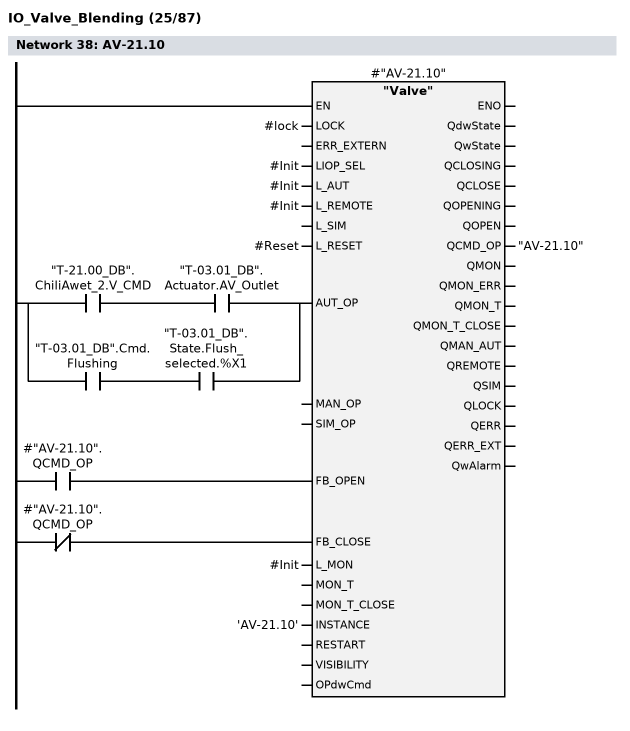
   RUNG wire#powerrail
      #"AV-21.10"(AUT_OP := wire#w1, FB_OPEN := wire#w2, FB_CLOSE := wire#w3, LOCK := #lock, ERR_EXTERN :=, LIOP_SEL := #Init, L_AUT := #Init, L_REMOTE := #Init, L_SIM :=, L_RESET := #Reset, MAN_OP :=, SIM_OP :=, L_MON := #Init, MON_T :=, MON_T_CLOSE :=, INSTANCE := 'AV-21.10', RESTART :=, VISIBILITY :=, OPdwCmd :=, QdwState =>, QwState =>, QCLOSING =>, QCLOSE =>, QOPENING =>, QOPEN =>, QCMD_OP => "AV-21.10", QMON =>, QMON_ERR =>, QMON_T =>, QMON_T_CLOSE =>, QMAN_AUT =>, QREMOTE =>, QSIM =>, QLOCK =>, QERR =>, QERR_EXT =>, QwAlarm =>)
   END_RUNG
   RUNG wire#powerrail
      Contact( "T-21.00_DB".ChiliAwet_2.V_CMD )
      Contact( "T-03.01_DB".Actuator.AV_Outlet )
   END_RUNG wire#w1
   RUNG wire#powerrail
      Contact( "T-03.01_DB".Cmd.Flushing )
      Contact( "T-03.01_DB".State.Flush_selected.%X1 )
   END_RUNG wire#w1
   RUNG wire#powerrail
      Contact( #"AV-21.10".QCMD_OP )
   END_RUNG wire#w2
   RUNG wire#powerrail
      I_Contact( #"AV-21.10".QCMD_OP )
   END_RUNG wire#w3
   // the same network as SCL:
   #"AV-21.10"(LOCK := #lock,   // "Valve"
               LIOP_SEL := #Init,
               L_AUT := #Init,
               L_REMOTE := #Init,
               L_RESET := #Reset,
               AUT_OP := ("T-21.00_DB".ChiliAwet_2.V_CMD AND "T-03.01_DB".Actuator.AV_Outlet) OR ("T-03.01_DB".Cmd.Flushing AND "T-03.01_DB".State.Flush_selected.%X1),
               FB_OPEN := #"AV-21.10".QCMD_OP,
               FB_CLOSE := NOT #"AV-21.10".QCMD_OP,
               L_MON := #Init,
               INSTANCE := 'AV-21.10',
               QCMD_OP => "AV-21.10");
END_REGION

REGION Network 39: AV-21.11
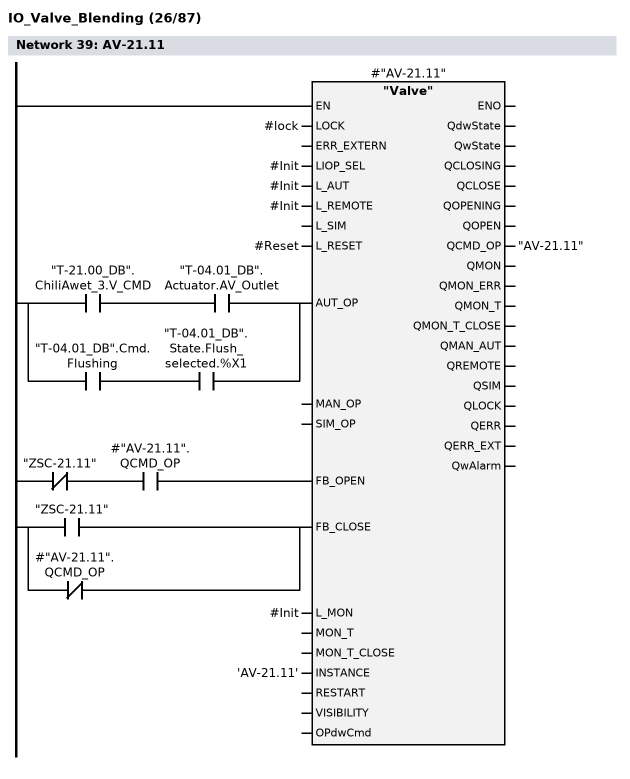
   RUNG wire#powerrail
      #"AV-21.11"(AUT_OP := wire#w1, FB_OPEN := wire#w2, FB_CLOSE := wire#w3, LOCK := #lock, ERR_EXTERN :=, LIOP_SEL := #Init, L_AUT := #Init, L_REMOTE := #Init, L_SIM :=, L_RESET := #Reset, MAN_OP :=, SIM_OP :=, L_MON := #Init, MON_T :=, MON_T_CLOSE :=, INSTANCE := 'AV-21.11', RESTART :=, VISIBILITY :=, OPdwCmd :=, QdwState =>, QwState =>, QCLOSING =>, QCLOSE =>, QOPENING =>, QOPEN =>, QCMD_OP => "AV-21.11", QMON =>, QMON_ERR =>, QMON_T =>, QMON_T_CLOSE =>, QMAN_AUT =>, QREMOTE =>, QSIM =>, QLOCK =>, QERR =>, QERR_EXT =>, QwAlarm =>)
   END_RUNG
   RUNG wire#powerrail
      Contact( "T-21.00_DB".ChiliAwet_3.V_CMD )
      Contact( "T-04.01_DB".Actuator.AV_Outlet )
   END_RUNG wire#w1
   RUNG wire#powerrail
      Contact( "T-04.01_DB".Cmd.Flushing )
      Contact( "T-04.01_DB".State.Flush_selected.%X1 )
   END_RUNG wire#w1
   RUNG wire#powerrail
      I_Contact( "ZSC-21.11" )
      Contact( #"AV-21.11".QCMD_OP )
   END_RUNG wire#w2
   RUNG wire#powerrail
      Contact( "ZSC-21.11" )
   END_RUNG wire#w3
   RUNG wire#powerrail
      I_Contact( #"AV-21.11".QCMD_OP )
   END_RUNG wire#w3
   // the same network as SCL:
   #"AV-21.11"(LOCK := #lock,   // "Valve"
               LIOP_SEL := #Init,
               L_AUT := #Init,
               L_REMOTE := #Init,
               L_RESET := #Reset,
               AUT_OP := ("T-21.00_DB".ChiliAwet_3.V_CMD AND "T-04.01_DB".Actuator.AV_Outlet) OR ("T-04.01_DB".Cmd.Flushing AND "T-04.01_DB".State.Flush_selected.%X1),
               FB_OPEN := NOT "ZSC-21.11" AND #"AV-21.11".QCMD_OP,
               FB_CLOSE := "ZSC-21.11" OR NOT #"AV-21.11".QCMD_OP,
               L_MON := #Init,
               INSTANCE := 'AV-21.11',
               QCMD_OP => "AV-21.11");
END_REGION

REGION Network 40: AV-21.12
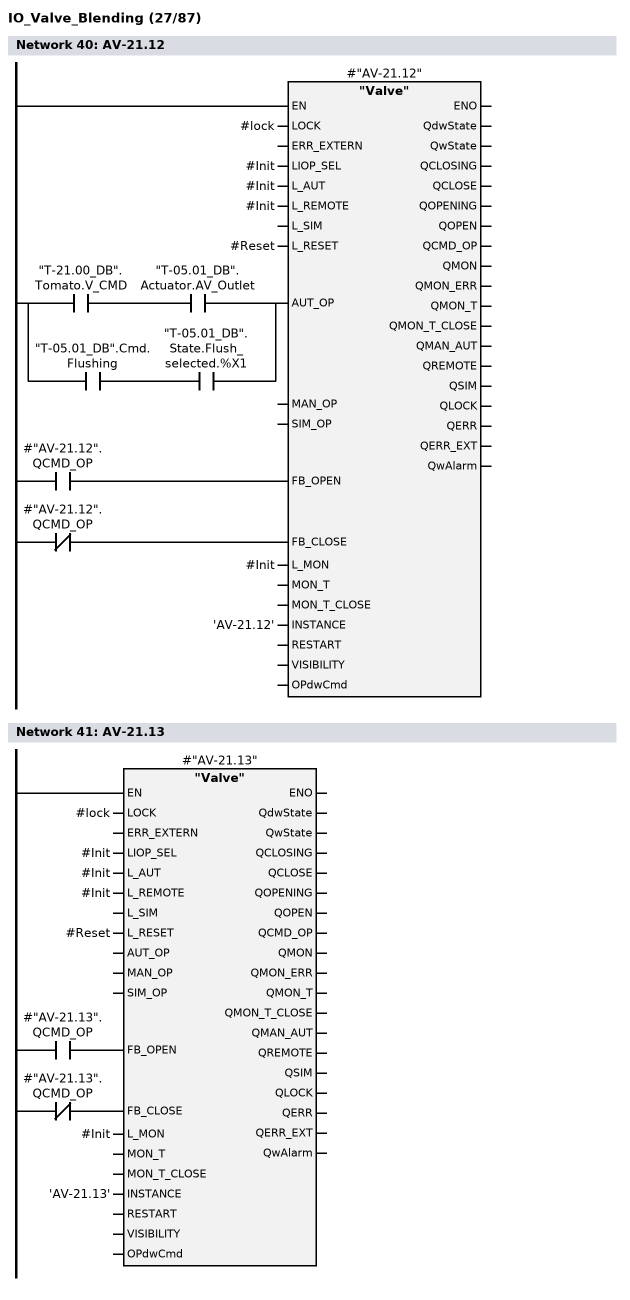
   RUNG wire#powerrail
      #"AV-21.12"(AUT_OP := wire#w1, FB_OPEN := wire#w2, FB_CLOSE := wire#w3, LOCK := #lock, ERR_EXTERN :=, LIOP_SEL := #Init, L_AUT := #Init, L_REMOTE := #Init, L_SIM :=, L_RESET := #Reset, MAN_OP :=, SIM_OP :=, L_MON := #Init, MON_T :=, MON_T_CLOSE :=, INSTANCE := 'AV-21.12', RESTART :=, VISIBILITY :=, OPdwCmd :=, QdwState =>, QwState =>, QCLOSING =>, QCLOSE =>, QOPENING =>, QOPEN =>, QCMD_OP =>, QMON =>, QMON_ERR =>, QMON_T =>, QMON_T_CLOSE =>, QMAN_AUT =>, QREMOTE =>, QSIM =>, QLOCK =>, QERR =>, QERR_EXT =>, QwAlarm =>)
   END_RUNG
   RUNG wire#powerrail
      Contact( "T-21.00_DB".Tomato.V_CMD )
      Contact( "T-05.01_DB".Actuator.AV_Outlet )
   END_RUNG wire#w1
   RUNG wire#powerrail
      Contact( "T-05.01_DB".Cmd.Flushing )
      Contact( "T-05.01_DB".State.Flush_selected.%X1 )
   END_RUNG wire#w1
   RUNG wire#powerrail
      Contact( #"AV-21.12".QCMD_OP )
   END_RUNG wire#w2
   RUNG wire#powerrail
      I_Contact( #"AV-21.12".QCMD_OP )
   END_RUNG wire#w3
   // the same network as SCL:
   #"AV-21.12"(LOCK := #lock,   // "Valve"
               LIOP_SEL := #Init,
               L_AUT := #Init,
               L_REMOTE := #Init,
               L_RESET := #Reset,
               AUT_OP := ("T-21.00_DB".Tomato.V_CMD AND "T-05.01_DB".Actuator.AV_Outlet) OR ("T-05.01_DB".Cmd.Flushing AND "T-05.01_DB".State.Flush_selected.%X1),
               FB_OPEN := #"AV-21.12".QCMD_OP,
               FB_CLOSE := NOT #"AV-21.12".QCMD_OP,
               L_MON := #Init,
               INSTANCE := 'AV-21.12');
END_REGION

REGION Network 41: AV-21.13
   RUNG wire#powerrail
      #"AV-21.13"(FB_OPEN := wire#w1, FB_CLOSE := wire#w2, LOCK := #lock, ERR_EXTERN :=, LIOP_SEL := #Init, L_AUT := #Init, L_REMOTE := #Init, L_SIM :=, L_RESET := #Reset, AUT_OP :=, MAN_OP :=, SIM_OP :=, L_MON := #Init, MON_T :=, MON_T_CLOSE :=, INSTANCE := 'AV-21.13', RESTART :=, VISIBILITY :=, OPdwCmd :=, QdwState =>, QwState =>, QCLOSING =>, QCLOSE =>, QOPENING =>, QOPEN =>, QCMD_OP =>, QMON =>, QMON_ERR =>, QMON_T =>, QMON_T_CLOSE =>, QMAN_AUT =>, QREMOTE =>, QSIM =>, QLOCK =>, QERR =>, QERR_EXT =>, QwAlarm =>)
   END_RUNG
   RUNG wire#powerrail
      Contact( #"AV-21.13".QCMD_OP )
   END_RUNG wire#w1
   RUNG wire#powerrail
      I_Contact( #"AV-21.13".QCMD_OP )
   END_RUNG wire#w2
   // the same network as SCL:
   #"AV-21.13"(LOCK := #lock,   // "Valve"
               LIOP_SEL := #Init,
               L_AUT := #Init,
               L_REMOTE := #Init,
               L_RESET := #Reset,
               FB_OPEN := #"AV-21.13".QCMD_OP,
               FB_CLOSE := NOT #"AV-21.13".QCMD_OP,
               L_MON := #Init,
               INSTANCE := 'AV-21.13');
END_REGION

REGION Network 42: AV-21.14
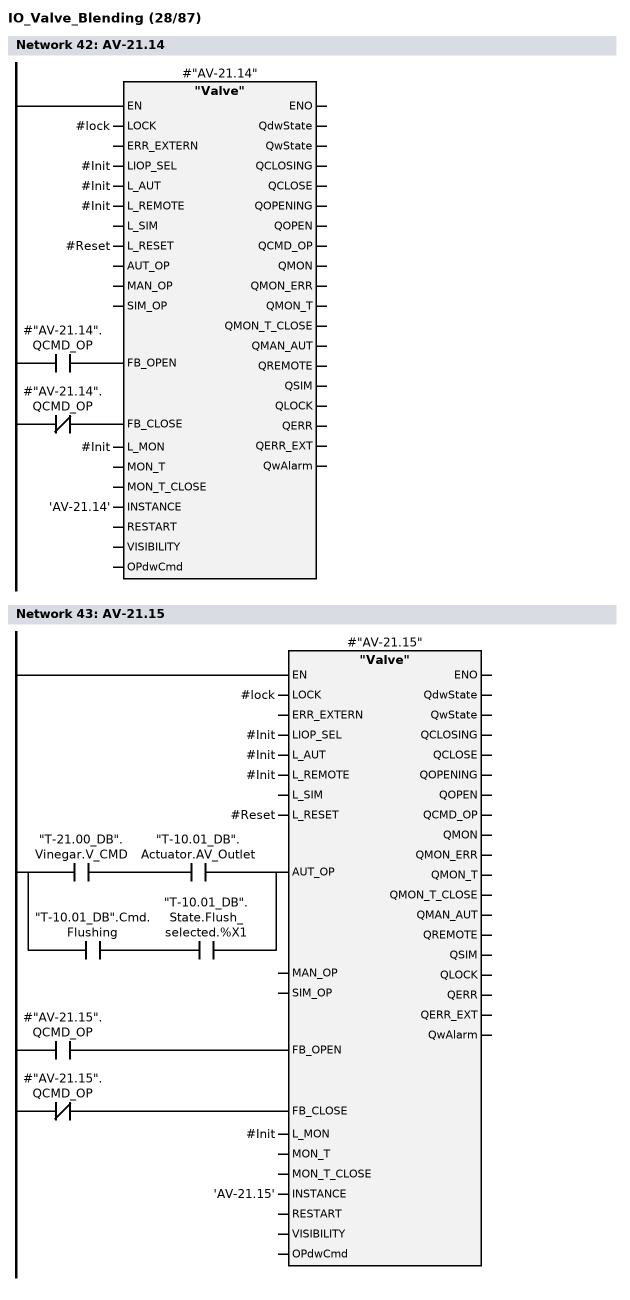
   RUNG wire#powerrail
      #"AV-21.14"(FB_OPEN := wire#w1, FB_CLOSE := wire#w2, LOCK := #lock, ERR_EXTERN :=, LIOP_SEL := #Init, L_AUT := #Init, L_REMOTE := #Init, L_SIM :=, L_RESET := #Reset, AUT_OP :=, MAN_OP :=, SIM_OP :=, L_MON := #Init, MON_T :=, MON_T_CLOSE :=, INSTANCE := 'AV-21.14', RESTART :=, VISIBILITY :=, OPdwCmd :=, QdwState =>, QwState =>, QCLOSING =>, QCLOSE =>, QOPENING =>, QOPEN =>, QCMD_OP =>, QMON =>, QMON_ERR =>, QMON_T =>, QMON_T_CLOSE =>, QMAN_AUT =>, QREMOTE =>, QSIM =>, QLOCK =>, QERR =>, QERR_EXT =>, QwAlarm =>)
   END_RUNG
   RUNG wire#powerrail
      Contact( #"AV-21.14".QCMD_OP )
   END_RUNG wire#w1
   RUNG wire#powerrail
      I_Contact( #"AV-21.14".QCMD_OP )
   END_RUNG wire#w2
   // the same network as SCL:
   #"AV-21.14"(LOCK := #lock,   // "Valve"
               LIOP_SEL := #Init,
               L_AUT := #Init,
               L_REMOTE := #Init,
               L_RESET := #Reset,
               FB_OPEN := #"AV-21.14".QCMD_OP,
               FB_CLOSE := NOT #"AV-21.14".QCMD_OP,
               L_MON := #Init,
               INSTANCE := 'AV-21.14');
END_REGION

REGION Network 43: AV-21.15
   RUNG wire#powerrail
      #"AV-21.15"(AUT_OP := wire#w1, FB_OPEN := wire#w2, FB_CLOSE := wire#w3, LOCK := #lock, ERR_EXTERN :=, LIOP_SEL := #Init, L_AUT := #Init, L_REMOTE := #Init, L_SIM :=, L_RESET := #Reset, MAN_OP :=, SIM_OP :=, L_MON := #Init, MON_T :=, MON_T_CLOSE :=, INSTANCE := 'AV-21.15', RESTART :=, VISIBILITY :=, OPdwCmd :=, QdwState =>, QwState =>, QCLOSING =>, QCLOSE =>, QOPENING =>, QOPEN =>, QCMD_OP =>, QMON =>, QMON_ERR =>, QMON_T =>, QMON_T_CLOSE =>, QMAN_AUT =>, QREMOTE =>, QSIM =>, QLOCK =>, QERR =>, QERR_EXT =>, QwAlarm =>)
   END_RUNG
   RUNG wire#powerrail
      Contact( "T-21.00_DB".Vinegar.V_CMD )
      Contact( "T-10.01_DB".Actuator.AV_Outlet )
   END_RUNG wire#w1
   RUNG wire#powerrail
      Contact( "T-10.01_DB".Cmd.Flushing )
      Contact( "T-10.01_DB".State.Flush_selected.%X1 )
   END_RUNG wire#w1
   RUNG wire#powerrail
      Contact( #"AV-21.15".QCMD_OP )
   END_RUNG wire#w2
   RUNG wire#powerrail
      I_Contact( #"AV-21.15".QCMD_OP )
   END_RUNG wire#w3
   // the same network as SCL:
   #"AV-21.15"(LOCK := #lock,   // "Valve"
               LIOP_SEL := #Init,
               L_AUT := #Init,
               L_REMOTE := #Init,
               L_RESET := #Reset,
               AUT_OP := ("T-21.00_DB".Vinegar.V_CMD AND "T-10.01_DB".Actuator.AV_Outlet) OR ("T-10.01_DB".Cmd.Flushing AND "T-10.01_DB".State.Flush_selected.%X1),
               FB_OPEN := #"AV-21.15".QCMD_OP,
               FB_CLOSE := NOT #"AV-21.15".QCMD_OP,
               L_MON := #Init,
               INSTANCE := 'AV-21.15');
END_REGION

REGION Network 44: AV-21.16
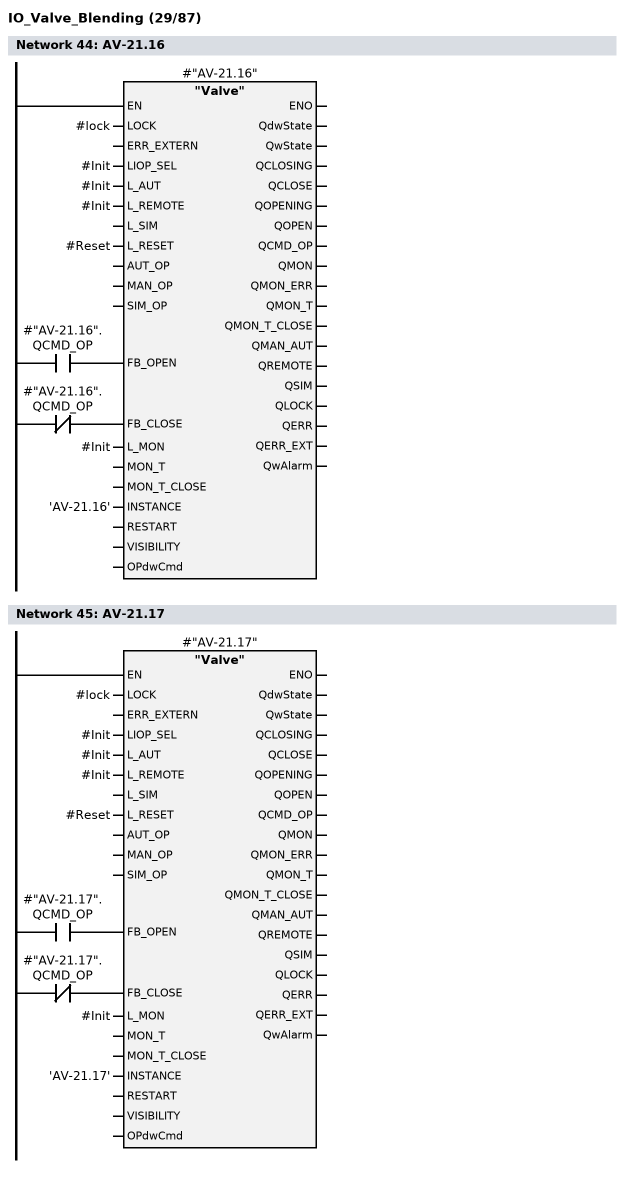
   RUNG wire#powerrail
      #"AV-21.16"(FB_OPEN := wire#w1, FB_CLOSE := wire#w2, LOCK := #lock, ERR_EXTERN :=, LIOP_SEL := #Init, L_AUT := #Init, L_REMOTE := #Init, L_SIM :=, L_RESET := #Reset, AUT_OP :=, MAN_OP :=, SIM_OP :=, L_MON := #Init, MON_T :=, MON_T_CLOSE :=, INSTANCE := 'AV-21.16', RESTART :=, VISIBILITY :=, OPdwCmd :=, QdwState =>, QwState =>, QCLOSING =>, QCLOSE =>, QOPENING =>, QOPEN =>, QCMD_OP =>, QMON =>, QMON_ERR =>, QMON_T =>, QMON_T_CLOSE =>, QMAN_AUT =>, QREMOTE =>, QSIM =>, QLOCK =>, QERR =>, QERR_EXT =>, QwAlarm =>)
   END_RUNG
   RUNG wire#powerrail
      Contact( #"AV-21.16".QCMD_OP )
   END_RUNG wire#w1
   RUNG wire#powerrail
      I_Contact( #"AV-21.16".QCMD_OP )
   END_RUNG wire#w2
   // the same network as SCL:
   #"AV-21.16"(LOCK := #lock,   // "Valve"
               LIOP_SEL := #Init,
               L_AUT := #Init,
               L_REMOTE := #Init,
               L_RESET := #Reset,
               FB_OPEN := #"AV-21.16".QCMD_OP,
               FB_CLOSE := NOT #"AV-21.16".QCMD_OP,
               L_MON := #Init,
               INSTANCE := 'AV-21.16');
END_REGION

REGION Network 45: AV-21.17
   RUNG wire#powerrail
      #"AV-21.17"(FB_OPEN := wire#w1, FB_CLOSE := wire#w2, LOCK := #lock, ERR_EXTERN :=, LIOP_SEL := #Init, L_AUT := #Init, L_REMOTE := #Init, L_SIM :=, L_RESET := #Reset, AUT_OP :=, MAN_OP :=, SIM_OP :=, L_MON := #Init, MON_T :=, MON_T_CLOSE :=, INSTANCE := 'AV-21.17', RESTART :=, VISIBILITY :=, OPdwCmd :=, QdwState =>, QwState =>, QCLOSING =>, QCLOSE =>, QOPENING =>, QOPEN =>, QCMD_OP =>, QMON =>, QMON_ERR =>, QMON_T =>, QMON_T_CLOSE =>, QMAN_AUT =>, QREMOTE =>, QSIM =>, QLOCK =>, QERR =>, QERR_EXT =>, QwAlarm =>)
   END_RUNG
   RUNG wire#powerrail
      Contact( #"AV-21.17".QCMD_OP )
   END_RUNG wire#w1
   RUNG wire#powerrail
      I_Contact( #"AV-21.17".QCMD_OP )
   END_RUNG wire#w2
   // the same network as SCL:
   #"AV-21.17"(LOCK := #lock,   // "Valve"
               LIOP_SEL := #Init,
               L_AUT := #Init,
               L_REMOTE := #Init,
               L_RESET := #Reset,
               FB_OPEN := #"AV-21.17".QCMD_OP,
               FB_CLOSE := NOT #"AV-21.17".QCMD_OP,
               L_MON := #Init,
               INSTANCE := 'AV-21.17');
END_REGION

REGION Network 46: AV-21.18
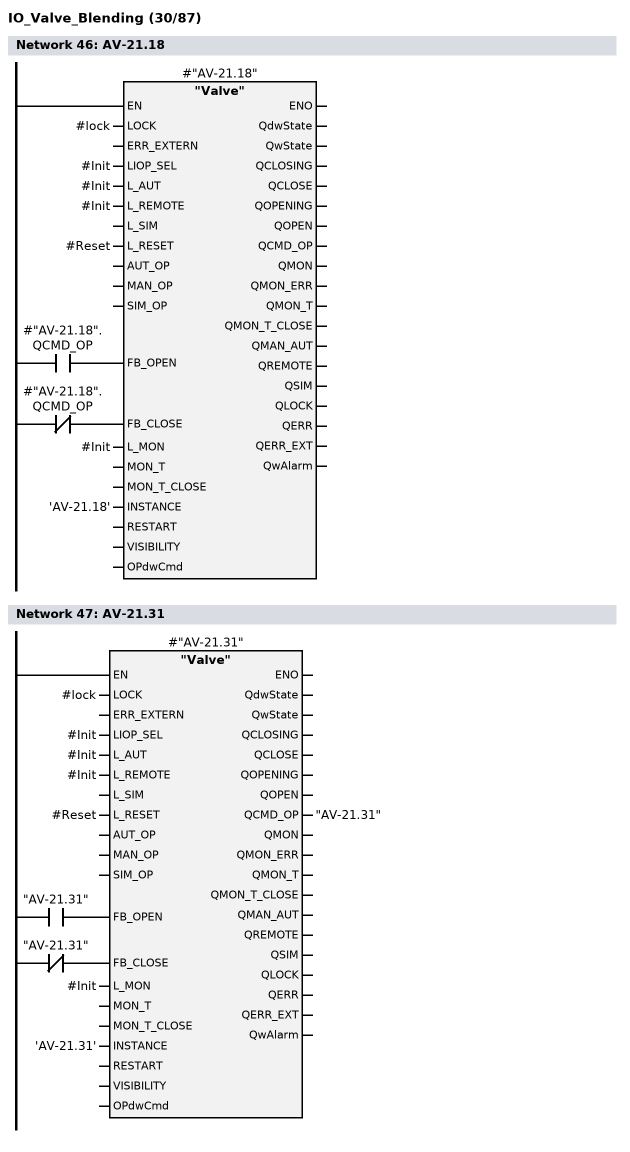
   RUNG wire#powerrail
      #"AV-21.18"(FB_OPEN := wire#w1, FB_CLOSE := wire#w2, LOCK := #lock, ERR_EXTERN :=, LIOP_SEL := #Init, L_AUT := #Init, L_REMOTE := #Init, L_SIM :=, L_RESET := #Reset, AUT_OP :=, MAN_OP :=, SIM_OP :=, L_MON := #Init, MON_T :=, MON_T_CLOSE :=, INSTANCE := 'AV-21.18', RESTART :=, VISIBILITY :=, OPdwCmd :=, QdwState =>, QwState =>, QCLOSING =>, QCLOSE =>, QOPENING =>, QOPEN =>, QCMD_OP =>, QMON =>, QMON_ERR =>, QMON_T =>, QMON_T_CLOSE =>, QMAN_AUT =>, QREMOTE =>, QSIM =>, QLOCK =>, QERR =>, QERR_EXT =>, QwAlarm =>)
   END_RUNG
   RUNG wire#powerrail
      Contact( #"AV-21.18".QCMD_OP )
   END_RUNG wire#w1
   RUNG wire#powerrail
      I_Contact( #"AV-21.18".QCMD_OP )
   END_RUNG wire#w2
   // the same network as SCL:
   #"AV-21.18"(LOCK := #lock,   // "Valve"
               LIOP_SEL := #Init,
               L_AUT := #Init,
               L_REMOTE := #Init,
               L_RESET := #Reset,
               FB_OPEN := #"AV-21.18".QCMD_OP,
               FB_CLOSE := NOT #"AV-21.18".QCMD_OP,
               L_MON := #Init,
               INSTANCE := 'AV-21.18');
END_REGION

REGION Network 47: AV-21.31
   RUNG wire#powerrail
      #"AV-21.31"(FB_OPEN := wire#w1, FB_CLOSE := wire#w2, LOCK := #lock, ERR_EXTERN :=, LIOP_SEL := #Init, L_AUT := #Init, L_REMOTE := #Init, L_SIM :=, L_RESET := #Reset, AUT_OP :=, MAN_OP :=, SIM_OP :=, L_MON := #Init, MON_T :=, MON_T_CLOSE :=, INSTANCE := 'AV-21.31', RESTART :=, VISIBILITY :=, OPdwCmd :=, QdwState =>, QwState =>, QCLOSING =>, QCLOSE =>, QOPENING =>, QOPEN =>, QCMD_OP => "AV-21.31", QMON =>, QMON_ERR =>, QMON_T =>, QMON_T_CLOSE =>, QMAN_AUT =>, QREMOTE =>, QSIM =>, QLOCK =>, QERR =>, QERR_EXT =>, QwAlarm =>)
   END_RUNG
   RUNG wire#powerrail
      Contact( "AV-21.31" )
   END_RUNG wire#w1
   RUNG wire#powerrail
      I_Contact( "AV-21.31" )
   END_RUNG wire#w2
   // the same network as SCL:
   #"AV-21.31"(LOCK := #lock,   // "Valve"
               LIOP_SEL := #Init,
               L_AUT := #Init,
               L_REMOTE := #Init,
               L_RESET := #Reset,
               FB_OPEN := "AV-21.31",
               FB_CLOSE := NOT "AV-21.31",
               L_MON := #Init,
               INSTANCE := 'AV-21.31',
               QCMD_OP => "AV-21.31");
END_REGION

REGION Network 48: AV-21.32
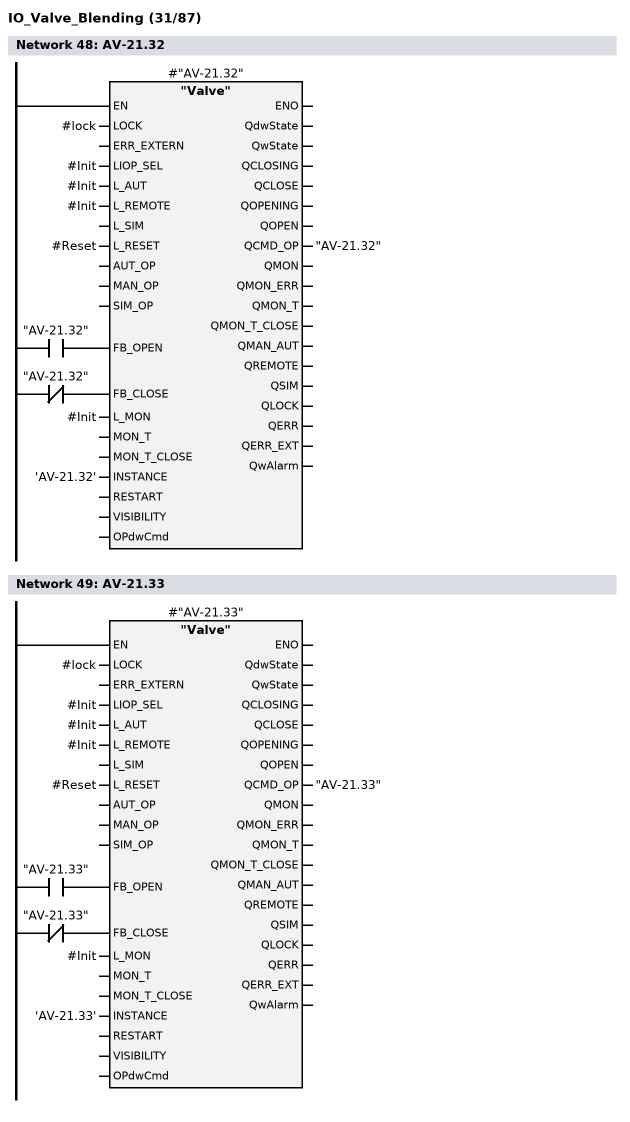
   RUNG wire#powerrail
      #"AV-21.32"(FB_OPEN := wire#w1, FB_CLOSE := wire#w2, LOCK := #lock, ERR_EXTERN :=, LIOP_SEL := #Init, L_AUT := #Init, L_REMOTE := #Init, L_SIM :=, L_RESET := #Reset, AUT_OP :=, MAN_OP :=, SIM_OP :=, L_MON := #Init, MON_T :=, MON_T_CLOSE :=, INSTANCE := 'AV-21.32', RESTART :=, VISIBILITY :=, OPdwCmd :=, QdwState =>, QwState =>, QCLOSING =>, QCLOSE =>, QOPENING =>, QOPEN =>, QCMD_OP => "AV-21.32", QMON =>, QMON_ERR =>, QMON_T =>, QMON_T_CLOSE =>, QMAN_AUT =>, QREMOTE =>, QSIM =>, QLOCK =>, QERR =>, QERR_EXT =>, QwAlarm =>)
   END_RUNG
   RUNG wire#powerrail
      Contact( "AV-21.32" )
   END_RUNG wire#w1
   RUNG wire#powerrail
      I_Contact( "AV-21.32" )
   END_RUNG wire#w2
   // the same network as SCL:
   #"AV-21.32"(LOCK := #lock,   // "Valve"
               LIOP_SEL := #Init,
               L_AUT := #Init,
               L_REMOTE := #Init,
               L_RESET := #Reset,
               FB_OPEN := "AV-21.32",
               FB_CLOSE := NOT "AV-21.32",
               L_MON := #Init,
               INSTANCE := 'AV-21.32',
               QCMD_OP => "AV-21.32");
END_REGION

REGION Network 49: AV-21.33
   RUNG wire#powerrail
      #"AV-21.33"(FB_OPEN := wire#w1, FB_CLOSE := wire#w2, LOCK := #lock, ERR_EXTERN :=, LIOP_SEL := #Init, L_AUT := #Init, L_REMOTE := #Init, L_SIM :=, L_RESET := #Reset, AUT_OP :=, MAN_OP :=, SIM_OP :=, L_MON := #Init, MON_T :=, MON_T_CLOSE :=, INSTANCE := 'AV-21.33', RESTART :=, VISIBILITY :=, OPdwCmd :=, QdwState =>, QwState =>, QCLOSING =>, QCLOSE =>, QOPENING =>, QOPEN =>, QCMD_OP => "AV-21.33", QMON =>, QMON_ERR =>, QMON_T =>, QMON_T_CLOSE =>, QMAN_AUT =>, QREMOTE =>, QSIM =>, QLOCK =>, QERR =>, QERR_EXT =>, QwAlarm =>)
   END_RUNG
   RUNG wire#powerrail
      Contact( "AV-21.33" )
   END_RUNG wire#w1
   RUNG wire#powerrail
      I_Contact( "AV-21.33" )
   END_RUNG wire#w2
   // the same network as SCL:
   #"AV-21.33"(LOCK := #lock,   // "Valve"
               LIOP_SEL := #Init,
               L_AUT := #Init,
               L_REMOTE := #Init,
               L_RESET := #Reset,
               FB_OPEN := "AV-21.33",
               FB_CLOSE := NOT "AV-21.33",
               L_MON := #Init,
               INSTANCE := 'AV-21.33',
               QCMD_OP => "AV-21.33");
END_REGION

REGION Network 50: AV-21.34
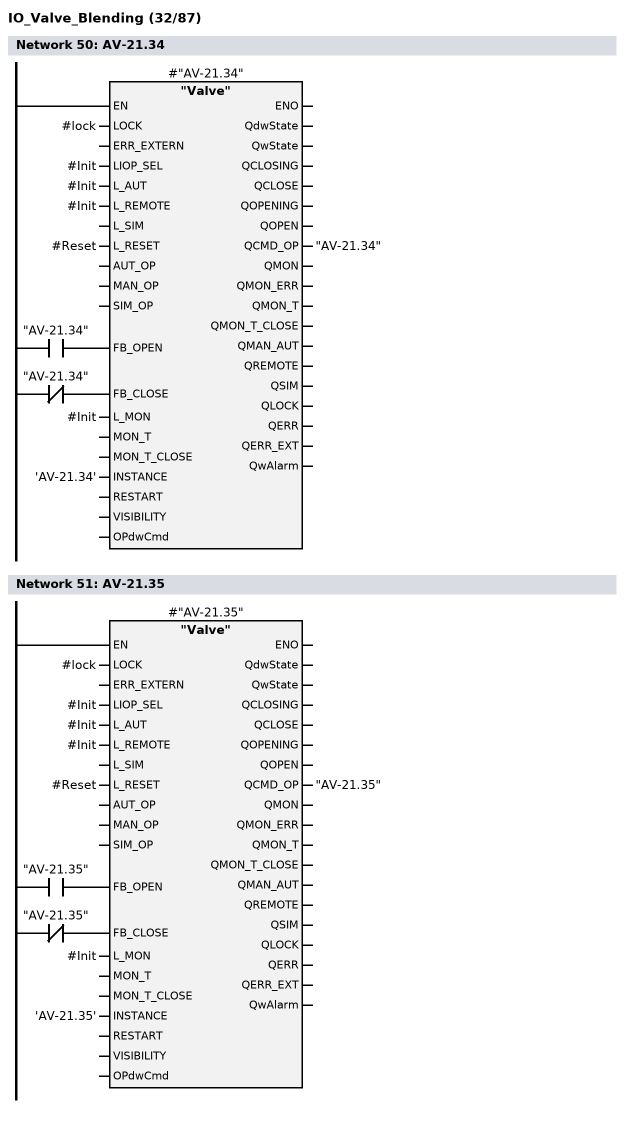
   RUNG wire#powerrail
      #"AV-21.34"(FB_OPEN := wire#w1, FB_CLOSE := wire#w2, LOCK := #lock, ERR_EXTERN :=, LIOP_SEL := #Init, L_AUT := #Init, L_REMOTE := #Init, L_SIM :=, L_RESET := #Reset, AUT_OP :=, MAN_OP :=, SIM_OP :=, L_MON := #Init, MON_T :=, MON_T_CLOSE :=, INSTANCE := 'AV-21.34', RESTART :=, VISIBILITY :=, OPdwCmd :=, QdwState =>, QwState =>, QCLOSING =>, QCLOSE =>, QOPENING =>, QOPEN =>, QCMD_OP => "AV-21.34", QMON =>, QMON_ERR =>, QMON_T =>, QMON_T_CLOSE =>, QMAN_AUT =>, QREMOTE =>, QSIM =>, QLOCK =>, QERR =>, QERR_EXT =>, QwAlarm =>)
   END_RUNG
   RUNG wire#powerrail
      Contact( "AV-21.34" )
   END_RUNG wire#w1
   RUNG wire#powerrail
      I_Contact( "AV-21.34" )
   END_RUNG wire#w2
   // the same network as SCL:
   #"AV-21.34"(LOCK := #lock,   // "Valve"
               LIOP_SEL := #Init,
               L_AUT := #Init,
               L_REMOTE := #Init,
               L_RESET := #Reset,
               FB_OPEN := "AV-21.34",
               FB_CLOSE := NOT "AV-21.34",
               L_MON := #Init,
               INSTANCE := 'AV-21.34',
               QCMD_OP => "AV-21.34");
END_REGION

REGION Network 51: AV-21.35
   RUNG wire#powerrail
      #"AV-21.35"(FB_OPEN := wire#w1, FB_CLOSE := wire#w2, LOCK := #lock, ERR_EXTERN :=, LIOP_SEL := #Init, L_AUT := #Init, L_REMOTE := #Init, L_SIM :=, L_RESET := #Reset, AUT_OP :=, MAN_OP :=, SIM_OP :=, L_MON := #Init, MON_T :=, MON_T_CLOSE :=, INSTANCE := 'AV-21.35', RESTART :=, VISIBILITY :=, OPdwCmd :=, QdwState =>, QwState =>, QCLOSING =>, QCLOSE =>, QOPENING =>, QOPEN =>, QCMD_OP => "AV-21.35", QMON =>, QMON_ERR =>, QMON_T =>, QMON_T_CLOSE =>, QMAN_AUT =>, QREMOTE =>, QSIM =>, QLOCK =>, QERR =>, QERR_EXT =>, QwAlarm =>)
   END_RUNG
   RUNG wire#powerrail
      Contact( "AV-21.35" )
   END_RUNG wire#w1
   RUNG wire#powerrail
      I_Contact( "AV-21.35" )
   END_RUNG wire#w2
   // the same network as SCL:
   #"AV-21.35"(LOCK := #lock,   // "Valve"
               LIOP_SEL := #Init,
               L_AUT := #Init,
               L_REMOTE := #Init,
               L_RESET := #Reset,
               FB_OPEN := "AV-21.35",
               FB_CLOSE := NOT "AV-21.35",
               L_MON := #Init,
               INSTANCE := 'AV-21.35',
               QCMD_OP => "AV-21.35");
END_REGION

REGION Network 52: AV-21.36
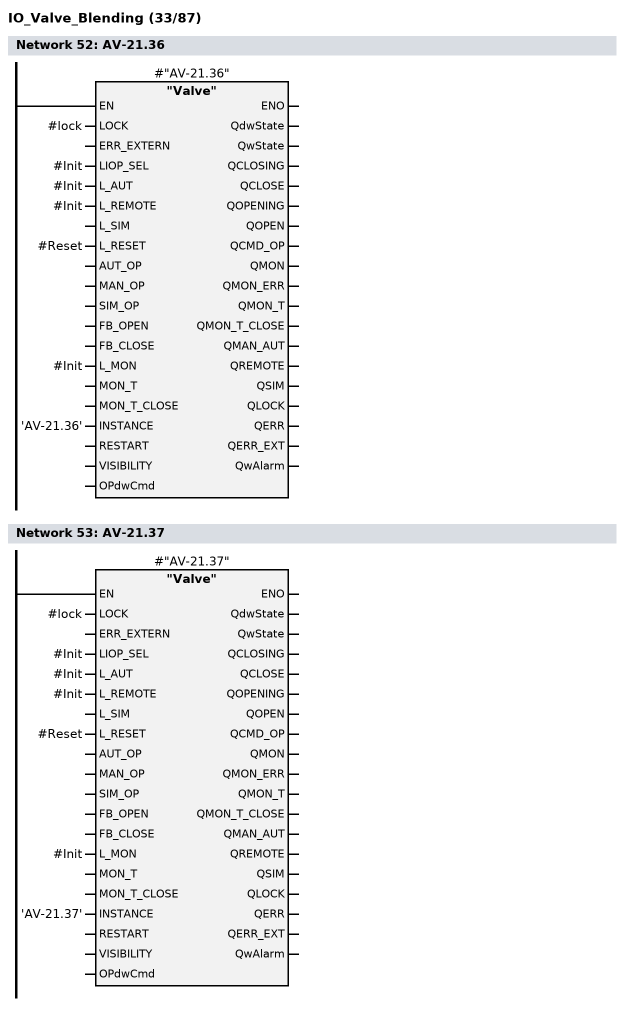
   RUNG wire#powerrail
      #"AV-21.36"(LOCK := #lock, ERR_EXTERN :=, LIOP_SEL := #Init, L_AUT := #Init, L_REMOTE := #Init, L_SIM :=, L_RESET := #Reset, AUT_OP :=, MAN_OP :=, SIM_OP :=, FB_OPEN :=, FB_CLOSE :=, L_MON := #Init, MON_T :=, MON_T_CLOSE :=, INSTANCE := 'AV-21.36', RESTART :=, VISIBILITY :=, OPdwCmd :=, QdwState =>, QwState =>, QCLOSING =>, QCLOSE =>, QOPENING =>, QOPEN =>, QCMD_OP =>, QMON =>, QMON_ERR =>, QMON_T =>, QMON_T_CLOSE =>, QMAN_AUT =>, QREMOTE =>, QSIM =>, QLOCK =>, QERR =>, QERR_EXT =>, QwAlarm =>)
   END_RUNG
   // the same network as SCL:
   #"AV-21.36"(LOCK := #lock,   // "Valve"
               LIOP_SEL := #Init,
               L_AUT := #Init,
               L_REMOTE := #Init,
               L_RESET := #Reset,
               L_MON := #Init,
               INSTANCE := 'AV-21.36');
END_REGION

REGION Network 53: AV-21.37
   RUNG wire#powerrail
      #"AV-21.37"(LOCK := #lock, ERR_EXTERN :=, LIOP_SEL := #Init, L_AUT := #Init, L_REMOTE := #Init, L_SIM :=, L_RESET := #Reset, AUT_OP :=, MAN_OP :=, SIM_OP :=, FB_OPEN :=, FB_CLOSE :=, L_MON := #Init, MON_T :=, MON_T_CLOSE :=, INSTANCE := 'AV-21.37', RESTART :=, VISIBILITY :=, OPdwCmd :=, QdwState =>, QwState =>, QCLOSING =>, QCLOSE =>, QOPENING =>, QOPEN =>, QCMD_OP =>, QMON =>, QMON_ERR =>, QMON_T =>, QMON_T_CLOSE =>, QMAN_AUT =>, QREMOTE =>, QSIM =>, QLOCK =>, QERR =>, QERR_EXT =>, QwAlarm =>)
   END_RUNG
   // the same network as SCL:
   #"AV-21.37"(LOCK := #lock,   // "Valve"
               LIOP_SEL := #Init,
               L_AUT := #Init,
               L_REMOTE := #Init,
               L_RESET := #Reset,
               L_MON := #Init,
               INSTANCE := 'AV-21.37');
END_REGION

REGION Network 54: AV-21.38
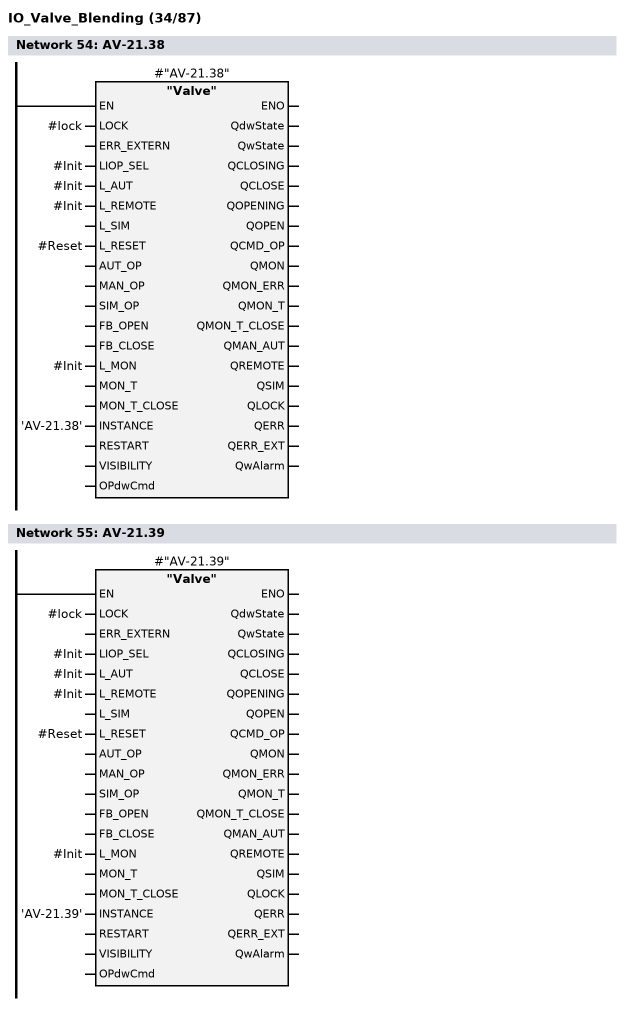
   RUNG wire#powerrail
      #"AV-21.38"(LOCK := #lock, ERR_EXTERN :=, LIOP_SEL := #Init, L_AUT := #Init, L_REMOTE := #Init, L_SIM :=, L_RESET := #Reset, AUT_OP :=, MAN_OP :=, SIM_OP :=, FB_OPEN :=, FB_CLOSE :=, L_MON := #Init, MON_T :=, MON_T_CLOSE :=, INSTANCE := 'AV-21.38', RESTART :=, VISIBILITY :=, OPdwCmd :=, QdwState =>, QwState =>, QCLOSING =>, QCLOSE =>, QOPENING =>, QOPEN =>, QCMD_OP =>, QMON =>, QMON_ERR =>, QMON_T =>, QMON_T_CLOSE =>, QMAN_AUT =>, QREMOTE =>, QSIM =>, QLOCK =>, QERR =>, QERR_EXT =>, QwAlarm =>)
   END_RUNG
   // the same network as SCL:
   #"AV-21.38"(LOCK := #lock,   // "Valve"
               LIOP_SEL := #Init,
               L_AUT := #Init,
               L_REMOTE := #Init,
               L_RESET := #Reset,
               L_MON := #Init,
               INSTANCE := 'AV-21.38');
END_REGION

REGION Network 55: AV-21.39
   RUNG wire#powerrail
      #"AV-21.39"(LOCK := #lock, ERR_EXTERN :=, LIOP_SEL := #Init, L_AUT := #Init, L_REMOTE := #Init, L_SIM :=, L_RESET := #Reset, AUT_OP :=, MAN_OP :=, SIM_OP :=, FB_OPEN :=, FB_CLOSE :=, L_MON := #Init, MON_T :=, MON_T_CLOSE :=, INSTANCE := 'AV-21.39', RESTART :=, VISIBILITY :=, OPdwCmd :=, QdwState =>, QwState =>, QCLOSING =>, QCLOSE =>, QOPENING =>, QOPEN =>, QCMD_OP =>, QMON =>, QMON_ERR =>, QMON_T =>, QMON_T_CLOSE =>, QMAN_AUT =>, QREMOTE =>, QSIM =>, QLOCK =>, QERR =>, QERR_EXT =>, QwAlarm =>)
   END_RUNG
   // the same network as SCL:
   #"AV-21.39"(LOCK := #lock,   // "Valve"
               LIOP_SEL := #Init,
               L_AUT := #Init,
               L_REMOTE := #Init,
               L_RESET := #Reset,
               L_MON := #Init,
               INSTANCE := 'AV-21.39');
END_REGION

REGION Network 56: AV-21.40
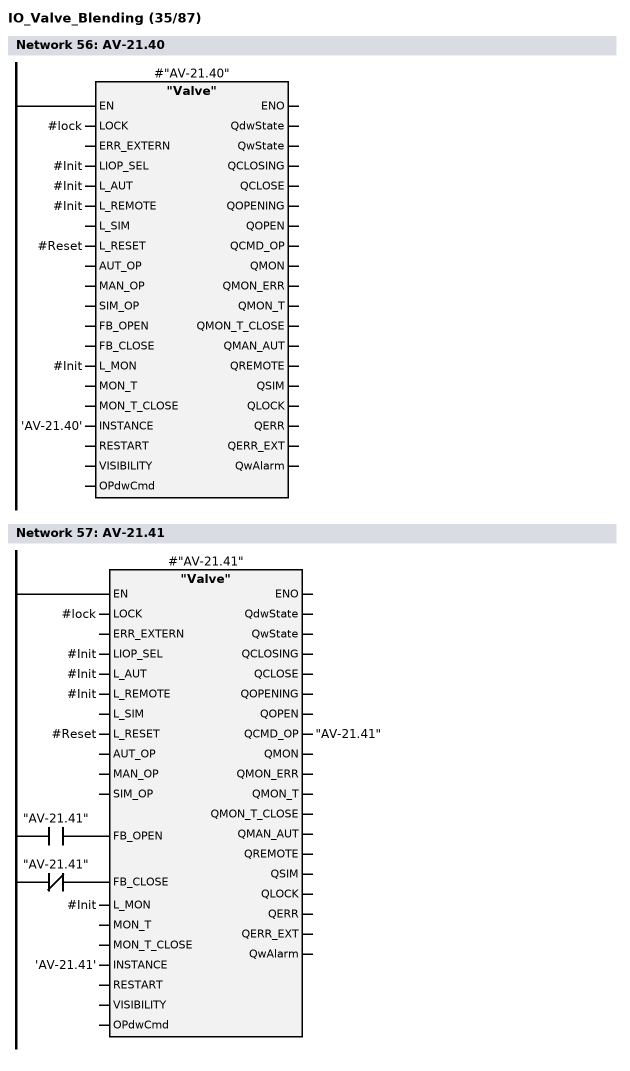
   RUNG wire#powerrail
      #"AV-21.40"(LOCK := #lock, ERR_EXTERN :=, LIOP_SEL := #Init, L_AUT := #Init, L_REMOTE := #Init, L_SIM :=, L_RESET := #Reset, AUT_OP :=, MAN_OP :=, SIM_OP :=, FB_OPEN :=, FB_CLOSE :=, L_MON := #Init, MON_T :=, MON_T_CLOSE :=, INSTANCE := 'AV-21.40', RESTART :=, VISIBILITY :=, OPdwCmd :=, QdwState =>, QwState =>, QCLOSING =>, QCLOSE =>, QOPENING =>, QOPEN =>, QCMD_OP =>, QMON =>, QMON_ERR =>, QMON_T =>, QMON_T_CLOSE =>, QMAN_AUT =>, QREMOTE =>, QSIM =>, QLOCK =>, QERR =>, QERR_EXT =>, QwAlarm =>)
   END_RUNG
   // the same network as SCL:
   #"AV-21.40"(LOCK := #lock,   // "Valve"
               LIOP_SEL := #Init,
               L_AUT := #Init,
               L_REMOTE := #Init,
               L_RESET := #Reset,
               L_MON := #Init,
               INSTANCE := 'AV-21.40');
END_REGION

REGION Network 57: AV-21.41
   RUNG wire#powerrail
      #"AV-21.41"(FB_OPEN := wire#w1, FB_CLOSE := wire#w2, LOCK := #lock, ERR_EXTERN :=, LIOP_SEL := #Init, L_AUT := #Init, L_REMOTE := #Init, L_SIM :=, L_RESET := #Reset, AUT_OP :=, MAN_OP :=, SIM_OP :=, L_MON := #Init, MON_T :=, MON_T_CLOSE :=, INSTANCE := 'AV-21.41', RESTART :=, VISIBILITY :=, OPdwCmd :=, QdwState =>, QwState =>, QCLOSING =>, QCLOSE =>, QOPENING =>, QOPEN =>, QCMD_OP => "AV-21.41", QMON =>, QMON_ERR =>, QMON_T =>, QMON_T_CLOSE =>, QMAN_AUT =>, QREMOTE =>, QSIM =>, QLOCK =>, QERR =>, QERR_EXT =>, QwAlarm =>)
   END_RUNG
   RUNG wire#powerrail
      Contact( "AV-21.41" )
   END_RUNG wire#w1
   RUNG wire#powerrail
      I_Contact( "AV-21.41" )
   END_RUNG wire#w2
   // the same network as SCL:
   #"AV-21.41"(LOCK := #lock,   // "Valve"
               LIOP_SEL := #Init,
               L_AUT := #Init,
               L_REMOTE := #Init,
               L_RESET := #Reset,
               FB_OPEN := "AV-21.41",
               FB_CLOSE := NOT "AV-21.41",
               L_MON := #Init,
               INSTANCE := 'AV-21.41',
               QCMD_OP => "AV-21.41");
END_REGION

REGION Network 58: AV-22.01
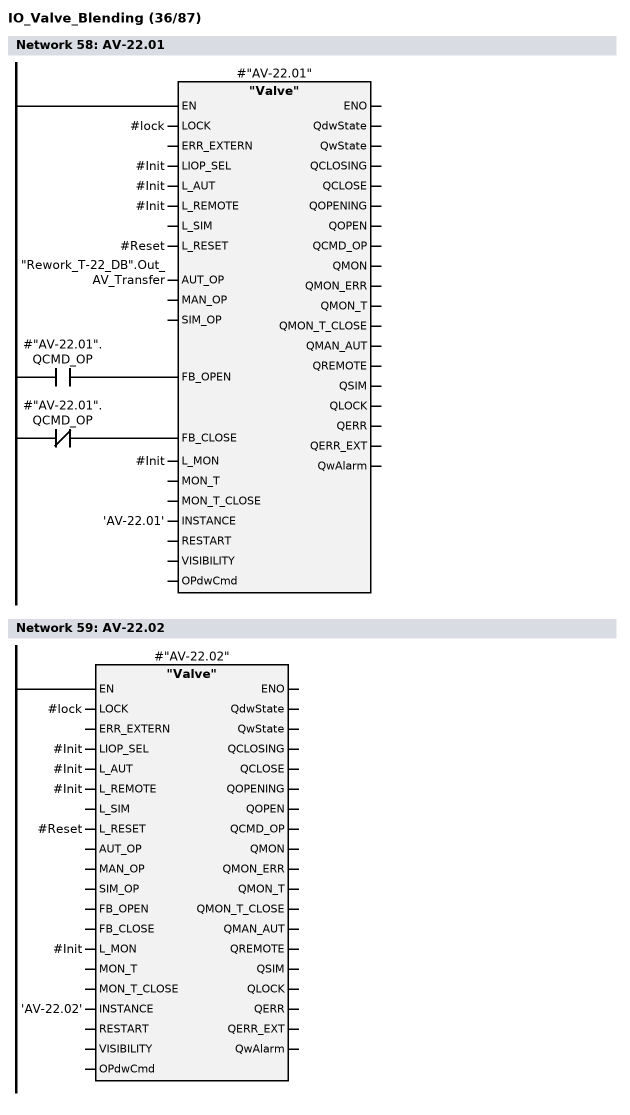
   RUNG wire#powerrail
      #"AV-22.01"(FB_OPEN := wire#w1, FB_CLOSE := wire#w2, LOCK := #lock, ERR_EXTERN :=, LIOP_SEL := #Init, L_AUT := #Init, L_REMOTE := #Init, L_SIM :=, L_RESET := #Reset, AUT_OP := "Rework_T-22_DB".Out_AV_Transfer, MAN_OP :=, SIM_OP :=, L_MON := #Init, MON_T :=, MON_T_CLOSE :=, INSTANCE := 'AV-22.01', RESTART :=, VISIBILITY :=, OPdwCmd :=, QdwState =>, QwState =>, QCLOSING =>, QCLOSE =>, QOPENING =>, QOPEN =>, QCMD_OP =>, QMON =>, QMON_ERR =>, QMON_T =>, QMON_T_CLOSE =>, QMAN_AUT =>, QREMOTE =>, QSIM =>, QLOCK =>, QERR =>, QERR_EXT =>, QwAlarm =>)
   END_RUNG
   RUNG wire#powerrail
      Contact( #"AV-22.01".QCMD_OP )
   END_RUNG wire#w1
   RUNG wire#powerrail
      I_Contact( #"AV-22.01".QCMD_OP )
   END_RUNG wire#w2
   // the same network as SCL:
   #"AV-22.01"(LOCK := #lock,   // "Valve"
               LIOP_SEL := #Init,
               L_AUT := #Init,
               L_REMOTE := #Init,
               L_RESET := #Reset,
               AUT_OP := "Rework_T-22_DB".Out_AV_Transfer,
               FB_OPEN := #"AV-22.01".QCMD_OP,
               FB_CLOSE := NOT #"AV-22.01".QCMD_OP,
               L_MON := #Init,
               INSTANCE := 'AV-22.01');
END_REGION

REGION Network 59: AV-22.02
   RUNG wire#powerrail
      #"AV-22.02"(LOCK := #lock, ERR_EXTERN :=, LIOP_SEL := #Init, L_AUT := #Init, L_REMOTE := #Init, L_SIM :=, L_RESET := #Reset, AUT_OP :=, MAN_OP :=, SIM_OP :=, FB_OPEN :=, FB_CLOSE :=, L_MON := #Init, MON_T :=, MON_T_CLOSE :=, INSTANCE := 'AV-22.02', RESTART :=, VISIBILITY :=, OPdwCmd :=, QdwState =>, QwState =>, QCLOSING =>, QCLOSE =>, QOPENING =>, QOPEN =>, QCMD_OP =>, QMON =>, QMON_ERR =>, QMON_T =>, QMON_T_CLOSE =>, QMAN_AUT =>, QREMOTE =>, QSIM =>, QLOCK =>, QERR =>, QERR_EXT =>, QwAlarm =>)
   END_RUNG
   // the same network as SCL:
   #"AV-22.02"(LOCK := #lock,   // "Valve"
               LIOP_SEL := #Init,
               L_AUT := #Init,
               L_REMOTE := #Init,
               L_RESET := #Reset,
               L_MON := #Init,
               INSTANCE := 'AV-22.02');
END_REGION

REGION Network 60: AV-22.03
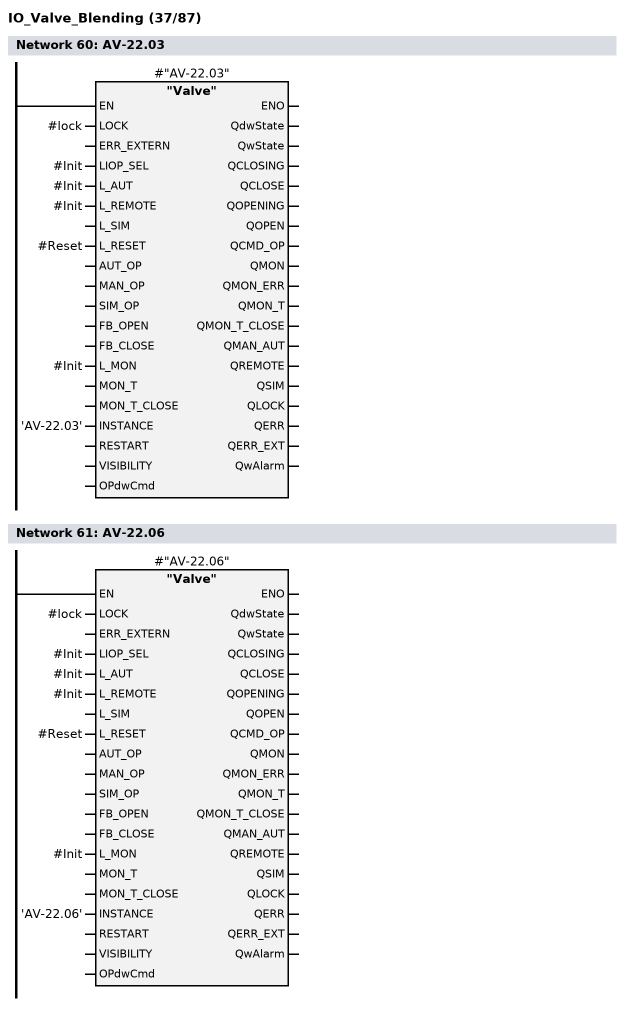
   RUNG wire#powerrail
      #"AV-22.03"(LOCK := #lock, ERR_EXTERN :=, LIOP_SEL := #Init, L_AUT := #Init, L_REMOTE := #Init, L_SIM :=, L_RESET := #Reset, AUT_OP :=, MAN_OP :=, SIM_OP :=, FB_OPEN :=, FB_CLOSE :=, L_MON := #Init, MON_T :=, MON_T_CLOSE :=, INSTANCE := 'AV-22.03', RESTART :=, VISIBILITY :=, OPdwCmd :=, QdwState =>, QwState =>, QCLOSING =>, QCLOSE =>, QOPENING =>, QOPEN =>, QCMD_OP =>, QMON =>, QMON_ERR =>, QMON_T =>, QMON_T_CLOSE =>, QMAN_AUT =>, QREMOTE =>, QSIM =>, QLOCK =>, QERR =>, QERR_EXT =>, QwAlarm =>)
   END_RUNG
   // the same network as SCL:
   #"AV-22.03"(LOCK := #lock,   // "Valve"
               LIOP_SEL := #Init,
               L_AUT := #Init,
               L_REMOTE := #Init,
               L_RESET := #Reset,
               L_MON := #Init,
               INSTANCE := 'AV-22.03');
END_REGION

REGION Network 61: AV-22.06
   RUNG wire#powerrail
      #"AV-22.06"(LOCK := #lock, ERR_EXTERN :=, LIOP_SEL := #Init, L_AUT := #Init, L_REMOTE := #Init, L_SIM :=, L_RESET := #Reset, AUT_OP :=, MAN_OP :=, SIM_OP :=, FB_OPEN :=, FB_CLOSE :=, L_MON := #Init, MON_T :=, MON_T_CLOSE :=, INSTANCE := 'AV-22.06', RESTART :=, VISIBILITY :=, OPdwCmd :=, QdwState =>, QwState =>, QCLOSING =>, QCLOSE =>, QOPENING =>, QOPEN =>, QCMD_OP =>, QMON =>, QMON_ERR =>, QMON_T =>, QMON_T_CLOSE =>, QMAN_AUT =>, QREMOTE =>, QSIM =>, QLOCK =>, QERR =>, QERR_EXT =>, QwAlarm =>)
   END_RUNG
   // the same network as SCL:
   #"AV-22.06"(LOCK := #lock,   // "Valve"
               LIOP_SEL := #Init,
               L_AUT := #Init,
               L_REMOTE := #Init,
               L_RESET := #Reset,
               L_MON := #Init,
               INSTANCE := 'AV-22.06');
END_REGION

REGION Network 62: AV-22.11
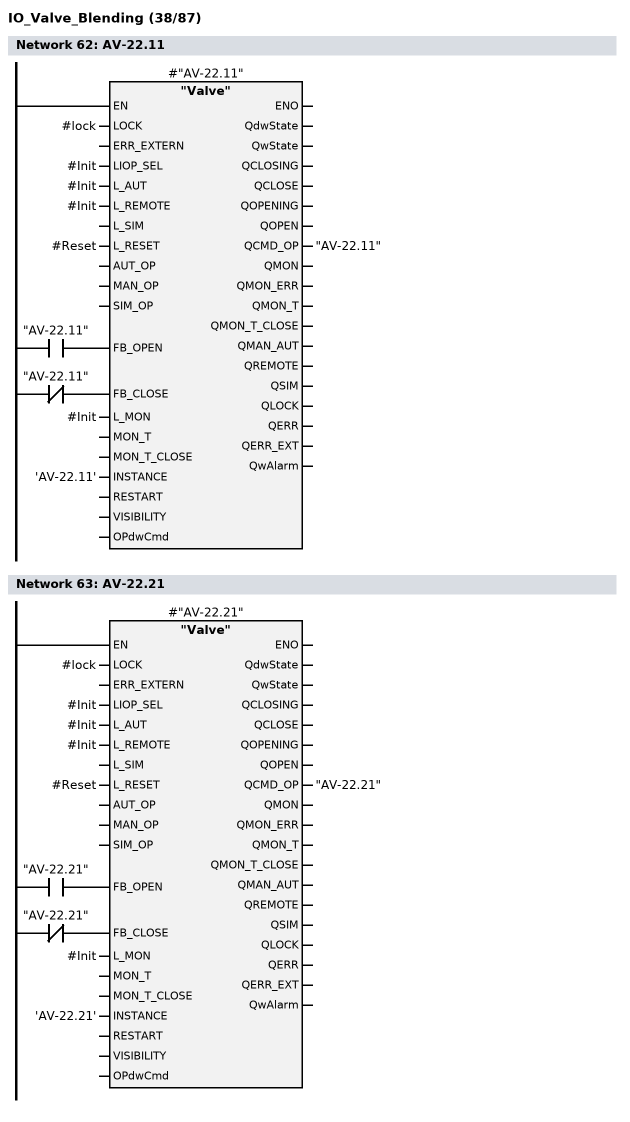
   RUNG wire#powerrail
      #"AV-22.11"(FB_OPEN := wire#w1, FB_CLOSE := wire#w2, LOCK := #lock, ERR_EXTERN :=, LIOP_SEL := #Init, L_AUT := #Init, L_REMOTE := #Init, L_SIM :=, L_RESET := #Reset, AUT_OP :=, MAN_OP :=, SIM_OP :=, L_MON := #Init, MON_T :=, MON_T_CLOSE :=, INSTANCE := 'AV-22.11', RESTART :=, VISIBILITY :=, OPdwCmd :=, QdwState =>, QwState =>, QCLOSING =>, QCLOSE =>, QOPENING =>, QOPEN =>, QCMD_OP => "AV-22.11", QMON =>, QMON_ERR =>, QMON_T =>, QMON_T_CLOSE =>, QMAN_AUT =>, QREMOTE =>, QSIM =>, QLOCK =>, QERR =>, QERR_EXT =>, QwAlarm =>)
   END_RUNG
   RUNG wire#powerrail
      Contact( "AV-22.11" )
   END_RUNG wire#w1
   RUNG wire#powerrail
      I_Contact( "AV-22.11" )
   END_RUNG wire#w2
   // the same network as SCL:
   #"AV-22.11"(LOCK := #lock,   // "Valve"
               LIOP_SEL := #Init,
               L_AUT := #Init,
               L_REMOTE := #Init,
               L_RESET := #Reset,
               FB_OPEN := "AV-22.11",
               FB_CLOSE := NOT "AV-22.11",
               L_MON := #Init,
               INSTANCE := 'AV-22.11',
               QCMD_OP => "AV-22.11");
END_REGION

REGION Network 63: AV-22.21
   RUNG wire#powerrail
      #"AV-22.21"(FB_OPEN := wire#w1, FB_CLOSE := wire#w2, LOCK := #lock, ERR_EXTERN :=, LIOP_SEL := #Init, L_AUT := #Init, L_REMOTE := #Init, L_SIM :=, L_RESET := #Reset, AUT_OP :=, MAN_OP :=, SIM_OP :=, L_MON := #Init, MON_T :=, MON_T_CLOSE :=, INSTANCE := 'AV-22.21', RESTART :=, VISIBILITY :=, OPdwCmd :=, QdwState =>, QwState =>, QCLOSING =>, QCLOSE =>, QOPENING =>, QOPEN =>, QCMD_OP => "AV-22.21", QMON =>, QMON_ERR =>, QMON_T =>, QMON_T_CLOSE =>, QMAN_AUT =>, QREMOTE =>, QSIM =>, QLOCK =>, QERR =>, QERR_EXT =>, QwAlarm =>)
   END_RUNG
   RUNG wire#powerrail
      Contact( "AV-22.21" )
   END_RUNG wire#w1
   RUNG wire#powerrail
      I_Contact( "AV-22.21" )
   END_RUNG wire#w2
   // the same network as SCL:
   #"AV-22.21"(LOCK := #lock,   // "Valve"
               LIOP_SEL := #Init,
               L_AUT := #Init,
               L_REMOTE := #Init,
               L_RESET := #Reset,
               FB_OPEN := "AV-22.21",
               FB_CLOSE := NOT "AV-22.21",
               L_MON := #Init,
               INSTANCE := 'AV-22.21',
               QCMD_OP => "AV-22.21");
END_REGION

REGION Network 64: AV-22.22
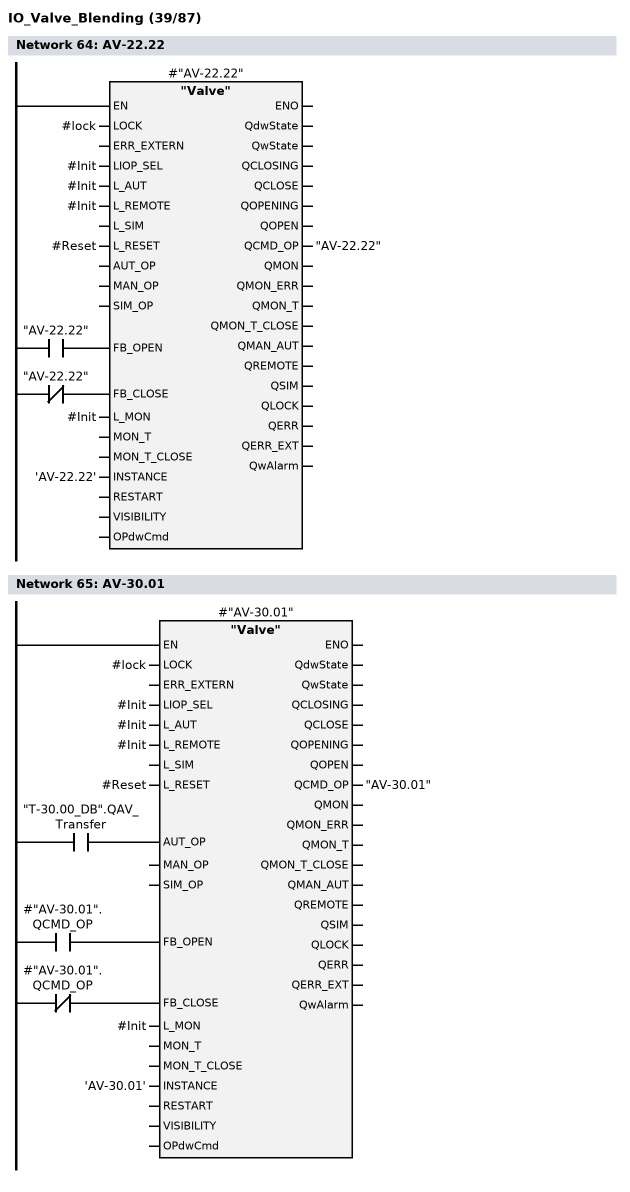
   RUNG wire#powerrail
      #"AV-22.22"(FB_OPEN := wire#w1, FB_CLOSE := wire#w2, LOCK := #lock, ERR_EXTERN :=, LIOP_SEL := #Init, L_AUT := #Init, L_REMOTE := #Init, L_SIM :=, L_RESET := #Reset, AUT_OP :=, MAN_OP :=, SIM_OP :=, L_MON := #Init, MON_T :=, MON_T_CLOSE :=, INSTANCE := 'AV-22.22', RESTART :=, VISIBILITY :=, OPdwCmd :=, QdwState =>, QwState =>, QCLOSING =>, QCLOSE =>, QOPENING =>, QOPEN =>, QCMD_OP => "AV-22.22", QMON =>, QMON_ERR =>, QMON_T =>, QMON_T_CLOSE =>, QMAN_AUT =>, QREMOTE =>, QSIM =>, QLOCK =>, QERR =>, QERR_EXT =>, QwAlarm =>)
   END_RUNG
   RUNG wire#powerrail
      Contact( "AV-22.22" )
   END_RUNG wire#w1
   RUNG wire#powerrail
      I_Contact( "AV-22.22" )
   END_RUNG wire#w2
   // the same network as SCL:
   #"AV-22.22"(LOCK := #lock,   // "Valve"
               LIOP_SEL := #Init,
               L_AUT := #Init,
               L_REMOTE := #Init,
               L_RESET := #Reset,
               FB_OPEN := "AV-22.22",
               FB_CLOSE := NOT "AV-22.22",
               L_MON := #Init,
               INSTANCE := 'AV-22.22',
               QCMD_OP => "AV-22.22");
END_REGION

REGION Network 65: AV-30.01
   RUNG wire#powerrail
      #"AV-30.01"(AUT_OP := wire#w1, FB_OPEN := wire#w2, FB_CLOSE := wire#w3, LOCK := #lock, ERR_EXTERN :=, LIOP_SEL := #Init, L_AUT := #Init, L_REMOTE := #Init, L_SIM :=, L_RESET := #Reset, MAN_OP :=, SIM_OP :=, L_MON := #Init, MON_T :=, MON_T_CLOSE :=, INSTANCE := 'AV-30.01', RESTART :=, VISIBILITY :=, OPdwCmd :=, QdwState =>, QwState =>, QCLOSING =>, QCLOSE =>, QOPENING =>, QOPEN =>, QCMD_OP => "AV-30.01", QMON =>, QMON_ERR =>, QMON_T =>, QMON_T_CLOSE =>, QMAN_AUT =>, QREMOTE =>, QSIM =>, QLOCK =>, QERR =>, QERR_EXT =>, QwAlarm =>)
   END_RUNG
   RUNG wire#powerrail
      Contact( "T-30.00_DB".QAV_Transfer )
   END_RUNG wire#w1
   RUNG wire#powerrail
      Contact( #"AV-30.01".QCMD_OP )
   END_RUNG wire#w2
   RUNG wire#powerrail
      I_Contact( #"AV-30.01".QCMD_OP )
   END_RUNG wire#w3
   // the same network as SCL:
   #"AV-30.01"(LOCK := #lock,   // "Valve"
               LIOP_SEL := #Init,
               L_AUT := #Init,
               L_REMOTE := #Init,
               L_RESET := #Reset,
               AUT_OP := "T-30.00_DB".QAV_Transfer,
               FB_OPEN := #"AV-30.01".QCMD_OP,
               FB_CLOSE := NOT #"AV-30.01".QCMD_OP,
               L_MON := #Init,
               INSTANCE := 'AV-30.01',
               QCMD_OP => "AV-30.01");
END_REGION

REGION Network 66: AV-30.02
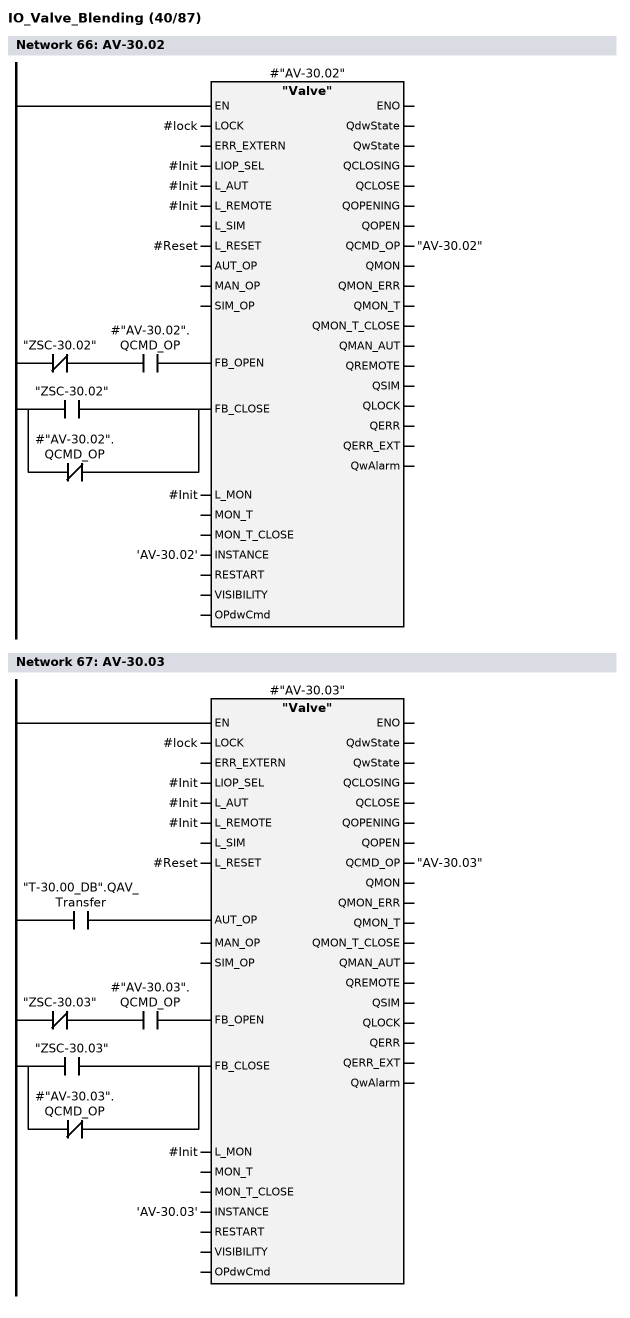
   RUNG wire#powerrail
      #"AV-30.02"(FB_OPEN := wire#w1, FB_CLOSE := wire#w2, LOCK := #lock, ERR_EXTERN :=, LIOP_SEL := #Init, L_AUT := #Init, L_REMOTE := #Init, L_SIM :=, L_RESET := #Reset, AUT_OP :=, MAN_OP :=, SIM_OP :=, L_MON := #Init, MON_T :=, MON_T_CLOSE :=, INSTANCE := 'AV-30.02', RESTART :=, VISIBILITY :=, OPdwCmd :=, QdwState =>, QwState =>, QCLOSING =>, QCLOSE =>, QOPENING =>, QOPEN =>, QCMD_OP => "AV-30.02", QMON =>, QMON_ERR =>, QMON_T =>, QMON_T_CLOSE =>, QMAN_AUT =>, QREMOTE =>, QSIM =>, QLOCK =>, QERR =>, QERR_EXT =>, QwAlarm =>)
   END_RUNG
   RUNG wire#powerrail
      I_Contact( "ZSC-30.02" )
      Contact( #"AV-30.02".QCMD_OP )
   END_RUNG wire#w1
   RUNG wire#powerrail
      Contact( "ZSC-30.02" )
   END_RUNG wire#w2
   RUNG wire#powerrail
      I_Contact( #"AV-30.02".QCMD_OP )
   END_RUNG wire#w2
   // the same network as SCL:
   #"AV-30.02"(LOCK := #lock,   // "Valve"
               LIOP_SEL := #Init,
               L_AUT := #Init,
               L_REMOTE := #Init,
               L_RESET := #Reset,
               FB_OPEN := NOT "ZSC-30.02" AND #"AV-30.02".QCMD_OP,
               FB_CLOSE := "ZSC-30.02" OR NOT #"AV-30.02".QCMD_OP,
               L_MON := #Init,
               INSTANCE := 'AV-30.02',
               QCMD_OP => "AV-30.02");
END_REGION

REGION Network 67: AV-30.03
   RUNG wire#powerrail
      #"AV-30.03"(AUT_OP := wire#w1, FB_OPEN := wire#w2, FB_CLOSE := wire#w3, LOCK := #lock, ERR_EXTERN :=, LIOP_SEL := #Init, L_AUT := #Init, L_REMOTE := #Init, L_SIM :=, L_RESET := #Reset, MAN_OP :=, SIM_OP :=, L_MON := #Init, MON_T :=, MON_T_CLOSE :=, INSTANCE := 'AV-30.03', RESTART :=, VISIBILITY :=, OPdwCmd :=, QdwState =>, QwState =>, QCLOSING =>, QCLOSE =>, QOPENING =>, QOPEN =>, QCMD_OP => "AV-30.03", QMON =>, QMON_ERR =>, QMON_T =>, QMON_T_CLOSE =>, QMAN_AUT =>, QREMOTE =>, QSIM =>, QLOCK =>, QERR =>, QERR_EXT =>, QwAlarm =>)
   END_RUNG
   RUNG wire#powerrail
      Contact( "T-30.00_DB".QAV_Transfer )
   END_RUNG wire#w1
   RUNG wire#powerrail
      I_Contact( "ZSC-30.03" )
      Contact( #"AV-30.03".QCMD_OP )
   END_RUNG wire#w2
   RUNG wire#powerrail
      Contact( "ZSC-30.03" )
   END_RUNG wire#w3
   RUNG wire#powerrail
      I_Contact( #"AV-30.03".QCMD_OP )
   END_RUNG wire#w3
   // the same network as SCL:
   #"AV-30.03"(LOCK := #lock,   // "Valve"
               LIOP_SEL := #Init,
               L_AUT := #Init,
               L_REMOTE := #Init,
               L_RESET := #Reset,
               AUT_OP := "T-30.00_DB".QAV_Transfer,
               FB_OPEN := NOT "ZSC-30.03" AND #"AV-30.03".QCMD_OP,
               FB_CLOSE := "ZSC-30.03" OR NOT #"AV-30.03".QCMD_OP,
               L_MON := #Init,
               INSTANCE := 'AV-30.03',
               QCMD_OP => "AV-30.03");
END_REGION

REGION Network 68: AV-30.04
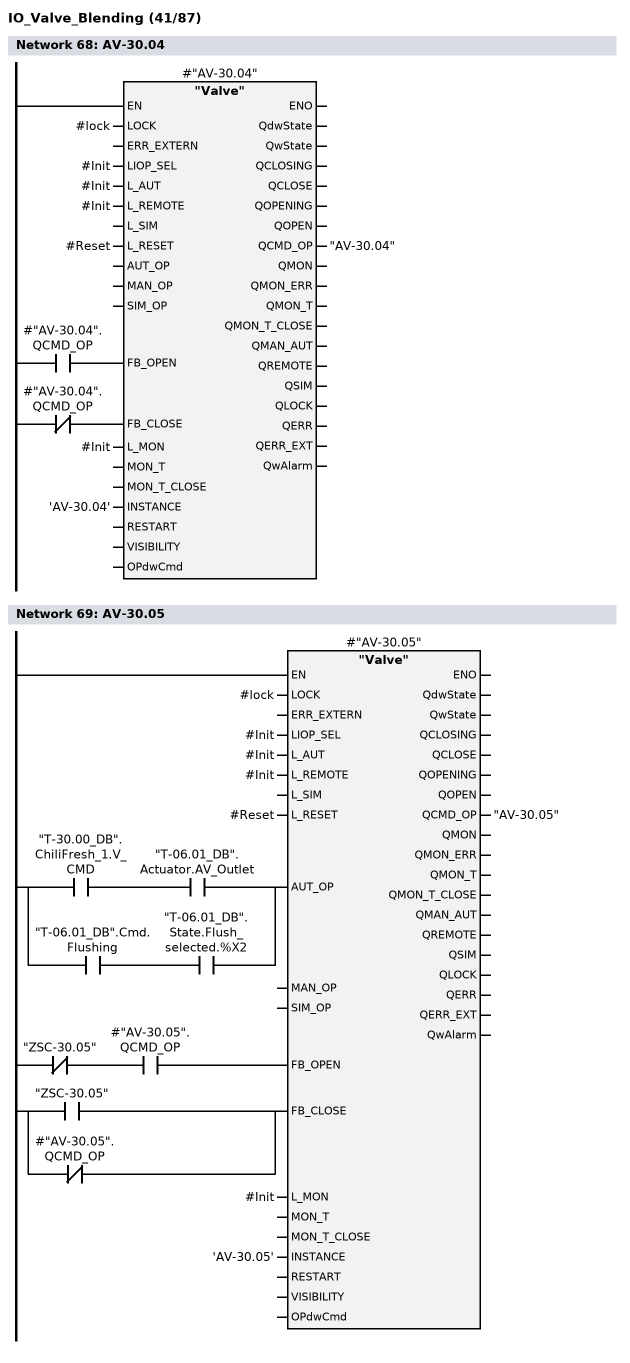
   RUNG wire#powerrail
      #"AV-30.04"(FB_OPEN := wire#w1, FB_CLOSE := wire#w2, LOCK := #lock, ERR_EXTERN :=, LIOP_SEL := #Init, L_AUT := #Init, L_REMOTE := #Init, L_SIM :=, L_RESET := #Reset, AUT_OP :=, MAN_OP :=, SIM_OP :=, L_MON := #Init, MON_T :=, MON_T_CLOSE :=, INSTANCE := 'AV-30.04', RESTART :=, VISIBILITY :=, OPdwCmd :=, QdwState =>, QwState =>, QCLOSING =>, QCLOSE =>, QOPENING =>, QOPEN =>, QCMD_OP => "AV-30.04", QMON =>, QMON_ERR =>, QMON_T =>, QMON_T_CLOSE =>, QMAN_AUT =>, QREMOTE =>, QSIM =>, QLOCK =>, QERR =>, QERR_EXT =>, QwAlarm =>)
   END_RUNG
   RUNG wire#powerrail
      Contact( #"AV-30.04".QCMD_OP )
   END_RUNG wire#w1
   RUNG wire#powerrail
      I_Contact( #"AV-30.04".QCMD_OP )
   END_RUNG wire#w2
   // the same network as SCL:
   #"AV-30.04"(LOCK := #lock,   // "Valve"
               LIOP_SEL := #Init,
               L_AUT := #Init,
               L_REMOTE := #Init,
               L_RESET := #Reset,
               FB_OPEN := #"AV-30.04".QCMD_OP,
               FB_CLOSE := NOT #"AV-30.04".QCMD_OP,
               L_MON := #Init,
               INSTANCE := 'AV-30.04',
               QCMD_OP => "AV-30.04");
END_REGION

REGION Network 69: AV-30.05
   RUNG wire#powerrail
      #"AV-30.05"(AUT_OP := wire#w1, FB_OPEN := wire#w2, FB_CLOSE := wire#w3, LOCK := #lock, ERR_EXTERN :=, LIOP_SEL := #Init, L_AUT := #Init, L_REMOTE := #Init, L_SIM :=, L_RESET := #Reset, MAN_OP :=, SIM_OP :=, L_MON := #Init, MON_T :=, MON_T_CLOSE :=, INSTANCE := 'AV-30.05', RESTART :=, VISIBILITY :=, OPdwCmd :=, QdwState =>, QwState =>, QCLOSING =>, QCLOSE =>, QOPENING =>, QOPEN =>, QCMD_OP => "AV-30.05", QMON =>, QMON_ERR =>, QMON_T =>, QMON_T_CLOSE =>, QMAN_AUT =>, QREMOTE =>, QSIM =>, QLOCK =>, QERR =>, QERR_EXT =>, QwAlarm =>)
   END_RUNG
   RUNG wire#powerrail
      Contact( "T-30.00_DB".ChiliFresh_1.V_CMD )
      Contact( "T-06.01_DB".Actuator.AV_Outlet )
   END_RUNG wire#w1
   RUNG wire#powerrail
      Contact( "T-06.01_DB".Cmd.Flushing )
      Contact( "T-06.01_DB".State.Flush_selected.%X2 )
   END_RUNG wire#w1
   RUNG wire#powerrail
      I_Contact( "ZSC-30.05" )
      Contact( #"AV-30.05".QCMD_OP )
   END_RUNG wire#w2
   RUNG wire#powerrail
      Contact( "ZSC-30.05" )
   END_RUNG wire#w3
   RUNG wire#powerrail
      I_Contact( #"AV-30.05".QCMD_OP )
   END_RUNG wire#w3
   // the same network as SCL:
   #"AV-30.05"(LOCK := #lock,   // "Valve"
               LIOP_SEL := #Init,
               L_AUT := #Init,
               L_REMOTE := #Init,
               L_RESET := #Reset,
               AUT_OP := ("T-30.00_DB".ChiliFresh_1.V_CMD AND "T-06.01_DB".Actuator.AV_Outlet) OR ("T-06.01_DB".Cmd.Flushing AND "T-06.01_DB".State.Flush_selected.%X2),
               FB_OPEN := NOT "ZSC-30.05" AND #"AV-30.05".QCMD_OP,
               FB_CLOSE := "ZSC-30.05" OR NOT #"AV-30.05".QCMD_OP,
               L_MON := #Init,
               INSTANCE := 'AV-30.05',
               QCMD_OP => "AV-30.05");
END_REGION

REGION Network 70: AV-30.06
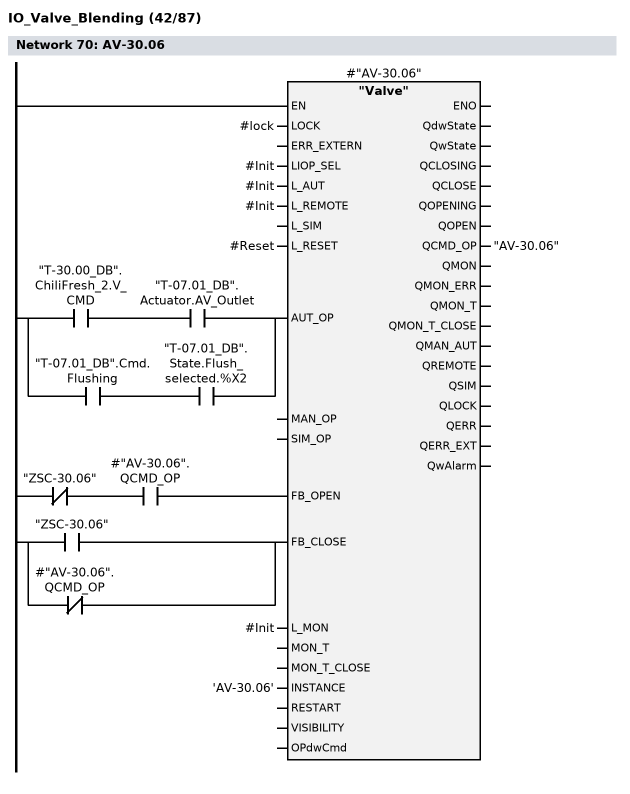
   RUNG wire#powerrail
      #"AV-30.06"(AUT_OP := wire#w1, FB_OPEN := wire#w2, FB_CLOSE := wire#w3, LOCK := #lock, ERR_EXTERN :=, LIOP_SEL := #Init, L_AUT := #Init, L_REMOTE := #Init, L_SIM :=, L_RESET := #Reset, MAN_OP :=, SIM_OP :=, L_MON := #Init, MON_T :=, MON_T_CLOSE :=, INSTANCE := 'AV-30.06', RESTART :=, VISIBILITY :=, OPdwCmd :=, QdwState =>, QwState =>, QCLOSING =>, QCLOSE =>, QOPENING =>, QOPEN =>, QCMD_OP => "AV-30.06", QMON =>, QMON_ERR =>, QMON_T =>, QMON_T_CLOSE =>, QMAN_AUT =>, QREMOTE =>, QSIM =>, QLOCK =>, QERR =>, QERR_EXT =>, QwAlarm =>)
   END_RUNG
   RUNG wire#powerrail
      Contact( "T-30.00_DB".ChiliFresh_2.V_CMD )
      Contact( "T-07.01_DB".Actuator.AV_Outlet )
   END_RUNG wire#w1
   RUNG wire#powerrail
      Contact( "T-07.01_DB".Cmd.Flushing )
      Contact( "T-07.01_DB".State.Flush_selected.%X2 )
   END_RUNG wire#w1
   RUNG wire#powerrail
      I_Contact( "ZSC-30.06" )
      Contact( #"AV-30.06".QCMD_OP )
   END_RUNG wire#w2
   RUNG wire#powerrail
      Contact( "ZSC-30.06" )
   END_RUNG wire#w3
   RUNG wire#powerrail
      I_Contact( #"AV-30.06".QCMD_OP )
   END_RUNG wire#w3
   // the same network as SCL:
   #"AV-30.06"(LOCK := #lock,   // "Valve"
               LIOP_SEL := #Init,
               L_AUT := #Init,
               L_REMOTE := #Init,
               L_RESET := #Reset,
               AUT_OP := ("T-30.00_DB".ChiliFresh_2.V_CMD AND "T-07.01_DB".Actuator.AV_Outlet) OR ("T-07.01_DB".Cmd.Flushing AND "T-07.01_DB".State.Flush_selected.%X2),
               FB_OPEN := NOT "ZSC-30.06" AND #"AV-30.06".QCMD_OP,
               FB_CLOSE := "ZSC-30.06" OR NOT #"AV-30.06".QCMD_OP,
               L_MON := #Init,
               INSTANCE := 'AV-30.06',
               QCMD_OP => "AV-30.06");
END_REGION

REGION Network 71: AV-30.07
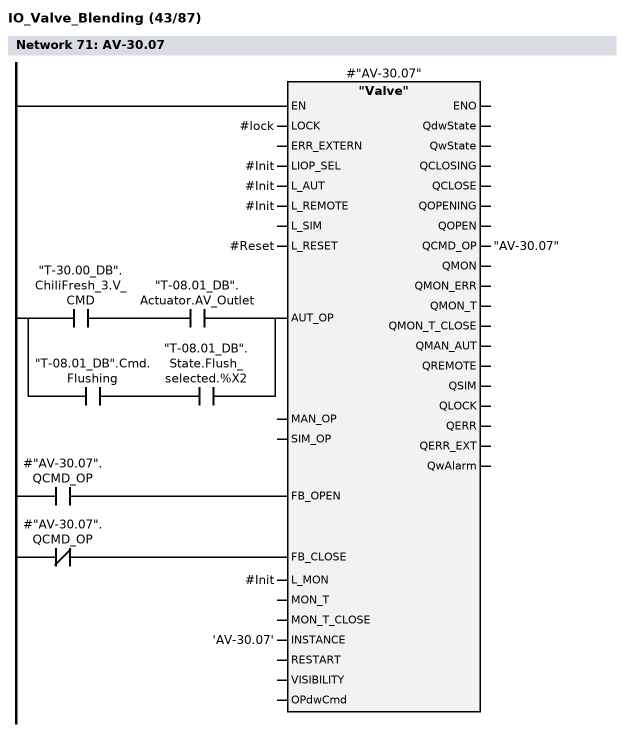
   RUNG wire#powerrail
      #"AV-30.07"(AUT_OP := wire#w1, FB_OPEN := wire#w2, FB_CLOSE := wire#w3, LOCK := #lock, ERR_EXTERN :=, LIOP_SEL := #Init, L_AUT := #Init, L_REMOTE := #Init, L_SIM :=, L_RESET := #Reset, MAN_OP :=, SIM_OP :=, L_MON := #Init, MON_T :=, MON_T_CLOSE :=, INSTANCE := 'AV-30.07', RESTART :=, VISIBILITY :=, OPdwCmd :=, QdwState =>, QwState =>, QCLOSING =>, QCLOSE =>, QOPENING =>, QOPEN =>, QCMD_OP => "AV-30.07", QMON =>, QMON_ERR =>, QMON_T =>, QMON_T_CLOSE =>, QMAN_AUT =>, QREMOTE =>, QSIM =>, QLOCK =>, QERR =>, QERR_EXT =>, QwAlarm =>)
   END_RUNG
   RUNG wire#powerrail
      Contact( "T-30.00_DB".ChiliFresh_3.V_CMD )
      Contact( "T-08.01_DB".Actuator.AV_Outlet )
   END_RUNG wire#w1
   RUNG wire#powerrail
      Contact( "T-08.01_DB".Cmd.Flushing )
      Contact( "T-08.01_DB".State.Flush_selected.%X2 )
   END_RUNG wire#w1
   RUNG wire#powerrail
      Contact( #"AV-30.07".QCMD_OP )
   END_RUNG wire#w2
   RUNG wire#powerrail
      I_Contact( #"AV-30.07".QCMD_OP )
   END_RUNG wire#w3
   // the same network as SCL:
   #"AV-30.07"(LOCK := #lock,   // "Valve"
               LIOP_SEL := #Init,
               L_AUT := #Init,
               L_REMOTE := #Init,
               L_RESET := #Reset,
               AUT_OP := ("T-30.00_DB".ChiliFresh_3.V_CMD AND "T-08.01_DB".Actuator.AV_Outlet) OR ("T-08.01_DB".Cmd.Flushing AND "T-08.01_DB".State.Flush_selected.%X2),
               FB_OPEN := #"AV-30.07".QCMD_OP,
               FB_CLOSE := NOT #"AV-30.07".QCMD_OP,
               L_MON := #Init,
               INSTANCE := 'AV-30.07',
               QCMD_OP => "AV-30.07");
END_REGION

REGION Network 72: AV-30.08
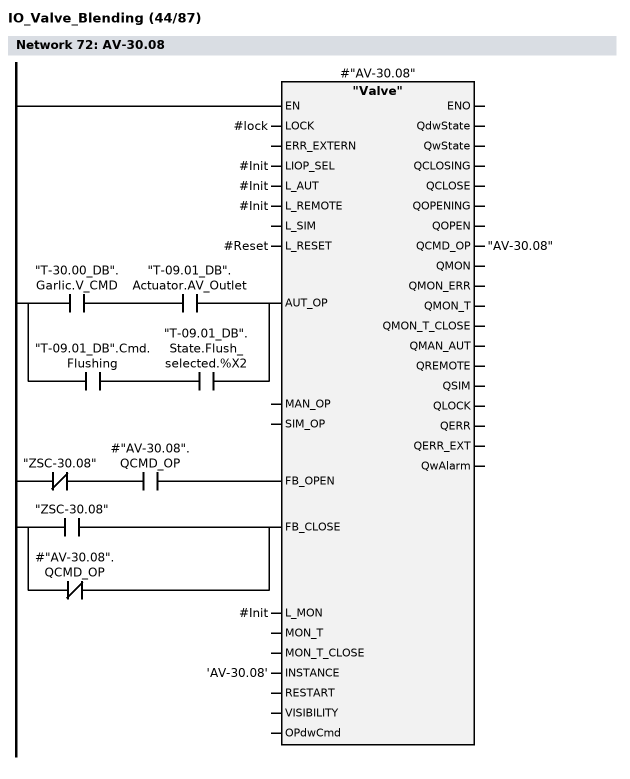
   RUNG wire#powerrail
      #"AV-30.08"(AUT_OP := wire#w1, FB_OPEN := wire#w2, FB_CLOSE := wire#w3, LOCK := #lock, ERR_EXTERN :=, LIOP_SEL := #Init, L_AUT := #Init, L_REMOTE := #Init, L_SIM :=, L_RESET := #Reset, MAN_OP :=, SIM_OP :=, L_MON := #Init, MON_T :=, MON_T_CLOSE :=, INSTANCE := 'AV-30.08', RESTART :=, VISIBILITY :=, OPdwCmd :=, QdwState =>, QwState =>, QCLOSING =>, QCLOSE =>, QOPENING =>, QOPEN =>, QCMD_OP => "AV-30.08", QMON =>, QMON_ERR =>, QMON_T =>, QMON_T_CLOSE =>, QMAN_AUT =>, QREMOTE =>, QSIM =>, QLOCK =>, QERR =>, QERR_EXT =>, QwAlarm =>)
   END_RUNG
   RUNG wire#powerrail
      Contact( "T-30.00_DB".Garlic.V_CMD )
      Contact( "T-09.01_DB".Actuator.AV_Outlet )
   END_RUNG wire#w1
   RUNG wire#powerrail
      Contact( "T-09.01_DB".Cmd.Flushing )
      Contact( "T-09.01_DB".State.Flush_selected.%X2 )
   END_RUNG wire#w1
   RUNG wire#powerrail
      I_Contact( "ZSC-30.08" )
      Contact( #"AV-30.08".QCMD_OP )
   END_RUNG wire#w2
   RUNG wire#powerrail
      Contact( "ZSC-30.08" )
   END_RUNG wire#w3
   RUNG wire#powerrail
      I_Contact( #"AV-30.08".QCMD_OP )
   END_RUNG wire#w3
   // the same network as SCL:
   #"AV-30.08"(LOCK := #lock,   // "Valve"
               LIOP_SEL := #Init,
               L_AUT := #Init,
               L_REMOTE := #Init,
               L_RESET := #Reset,
               AUT_OP := ("T-30.00_DB".Garlic.V_CMD AND "T-09.01_DB".Actuator.AV_Outlet) OR ("T-09.01_DB".Cmd.Flushing AND "T-09.01_DB".State.Flush_selected.%X2),
               FB_OPEN := NOT "ZSC-30.08" AND #"AV-30.08".QCMD_OP,
               FB_CLOSE := "ZSC-30.08" OR NOT #"AV-30.08".QCMD_OP,
               L_MON := #Init,
               INSTANCE := 'AV-30.08',
               QCMD_OP => "AV-30.08");
END_REGION

REGION Network 73: AV-30.09
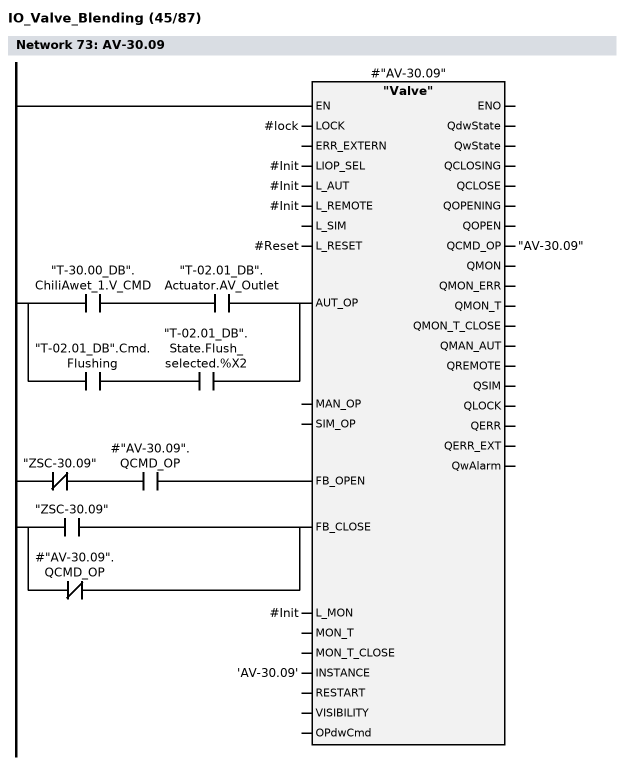
   RUNG wire#powerrail
      #"AV-30.09"(AUT_OP := wire#w1, FB_OPEN := wire#w2, FB_CLOSE := wire#w3, LOCK := #lock, ERR_EXTERN :=, LIOP_SEL := #Init, L_AUT := #Init, L_REMOTE := #Init, L_SIM :=, L_RESET := #Reset, MAN_OP :=, SIM_OP :=, L_MON := #Init, MON_T :=, MON_T_CLOSE :=, INSTANCE := 'AV-30.09', RESTART :=, VISIBILITY :=, OPdwCmd :=, QdwState =>, QwState =>, QCLOSING =>, QCLOSE =>, QOPENING =>, QOPEN =>, QCMD_OP => "AV-30.09", QMON =>, QMON_ERR =>, QMON_T =>, QMON_T_CLOSE =>, QMAN_AUT =>, QREMOTE =>, QSIM =>, QLOCK =>, QERR =>, QERR_EXT =>, QwAlarm =>)
   END_RUNG
   RUNG wire#powerrail
      Contact( "T-30.00_DB".ChiliAwet_1.V_CMD )
      Contact( "T-02.01_DB".Actuator.AV_Outlet )
   END_RUNG wire#w1
   RUNG wire#powerrail
      Contact( "T-02.01_DB".Cmd.Flushing )
      Contact( "T-02.01_DB".State.Flush_selected.%X2 )
   END_RUNG wire#w1
   RUNG wire#powerrail
      I_Contact( "ZSC-30.09" )
      Contact( #"AV-30.09".QCMD_OP )
   END_RUNG wire#w2
   RUNG wire#powerrail
      Contact( "ZSC-30.09" )
   END_RUNG wire#w3
   RUNG wire#powerrail
      I_Contact( #"AV-30.09".QCMD_OP )
   END_RUNG wire#w3
   // the same network as SCL:
   #"AV-30.09"(LOCK := #lock,   // "Valve"
               LIOP_SEL := #Init,
               L_AUT := #Init,
               L_REMOTE := #Init,
               L_RESET := #Reset,
               AUT_OP := ("T-30.00_DB".ChiliAwet_1.V_CMD AND "T-02.01_DB".Actuator.AV_Outlet) OR ("T-02.01_DB".Cmd.Flushing AND "T-02.01_DB".State.Flush_selected.%X2),
               FB_OPEN := NOT "ZSC-30.09" AND #"AV-30.09".QCMD_OP,
               FB_CLOSE := "ZSC-30.09" OR NOT #"AV-30.09".QCMD_OP,
               L_MON := #Init,
               INSTANCE := 'AV-30.09',
               QCMD_OP => "AV-30.09");
END_REGION

REGION Network 74: AV-30.10
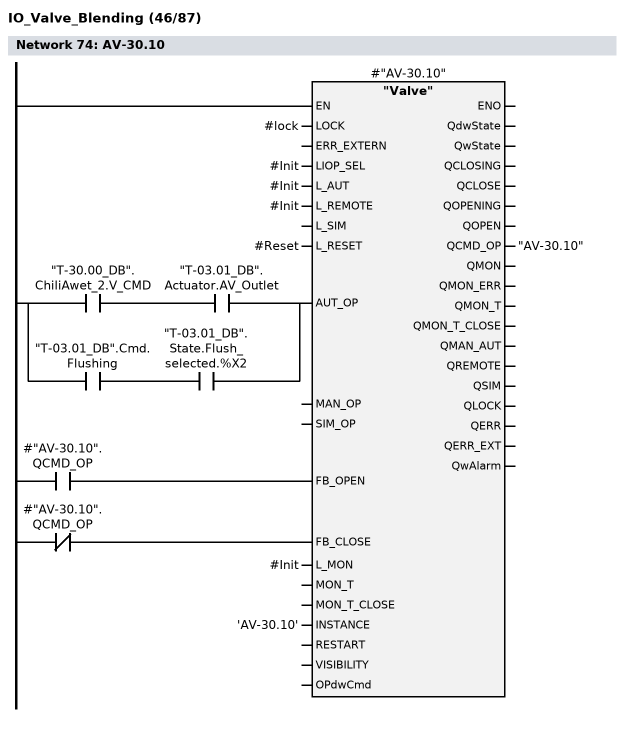
   RUNG wire#powerrail
      #"AV-30.10"(AUT_OP := wire#w1, FB_OPEN := wire#w2, FB_CLOSE := wire#w3, LOCK := #lock, ERR_EXTERN :=, LIOP_SEL := #Init, L_AUT := #Init, L_REMOTE := #Init, L_SIM :=, L_RESET := #Reset, MAN_OP :=, SIM_OP :=, L_MON := #Init, MON_T :=, MON_T_CLOSE :=, INSTANCE := 'AV-30.10', RESTART :=, VISIBILITY :=, OPdwCmd :=, QdwState =>, QwState =>, QCLOSING =>, QCLOSE =>, QOPENING =>, QOPEN =>, QCMD_OP => "AV-30.10", QMON =>, QMON_ERR =>, QMON_T =>, QMON_T_CLOSE =>, QMAN_AUT =>, QREMOTE =>, QSIM =>, QLOCK =>, QERR =>, QERR_EXT =>, QwAlarm =>)
   END_RUNG
   RUNG wire#powerrail
      Contact( "T-30.00_DB".ChiliAwet_2.V_CMD )
      Contact( "T-03.01_DB".Actuator.AV_Outlet )
   END_RUNG wire#w1
   RUNG wire#powerrail
      Contact( "T-03.01_DB".Cmd.Flushing )
      Contact( "T-03.01_DB".State.Flush_selected.%X2 )
   END_RUNG wire#w1
   RUNG wire#powerrail
      Contact( #"AV-30.10".QCMD_OP )
   END_RUNG wire#w2
   RUNG wire#powerrail
      I_Contact( #"AV-30.10".QCMD_OP )
   END_RUNG wire#w3
   // the same network as SCL:
   #"AV-30.10"(LOCK := #lock,   // "Valve"
               LIOP_SEL := #Init,
               L_AUT := #Init,
               L_REMOTE := #Init,
               L_RESET := #Reset,
               AUT_OP := ("T-30.00_DB".ChiliAwet_2.V_CMD AND "T-03.01_DB".Actuator.AV_Outlet) OR ("T-03.01_DB".Cmd.Flushing AND "T-03.01_DB".State.Flush_selected.%X2),
               FB_OPEN := #"AV-30.10".QCMD_OP,
               FB_CLOSE := NOT #"AV-30.10".QCMD_OP,
               L_MON := #Init,
               INSTANCE := 'AV-30.10',
               QCMD_OP => "AV-30.10");
END_REGION

REGION Network 75: AV-30.11
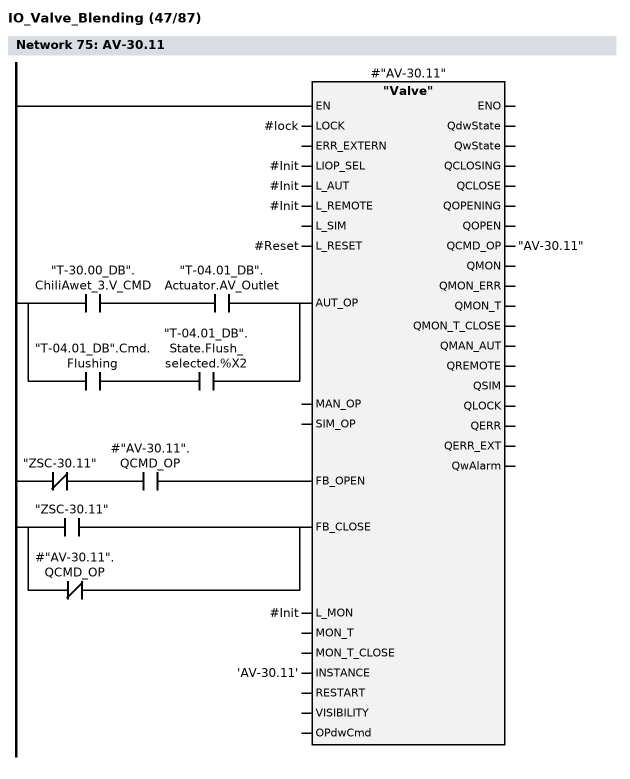
   RUNG wire#powerrail
      #"AV-30.11"(AUT_OP := wire#w1, FB_OPEN := wire#w2, FB_CLOSE := wire#w3, LOCK := #lock, ERR_EXTERN :=, LIOP_SEL := #Init, L_AUT := #Init, L_REMOTE := #Init, L_SIM :=, L_RESET := #Reset, MAN_OP :=, SIM_OP :=, L_MON := #Init, MON_T :=, MON_T_CLOSE :=, INSTANCE := 'AV-30.11', RESTART :=, VISIBILITY :=, OPdwCmd :=, QdwState =>, QwState =>, QCLOSING =>, QCLOSE =>, QOPENING =>, QOPEN =>, QCMD_OP => "AV-30.11", QMON =>, QMON_ERR =>, QMON_T =>, QMON_T_CLOSE =>, QMAN_AUT =>, QREMOTE =>, QSIM =>, QLOCK =>, QERR =>, QERR_EXT =>, QwAlarm =>)
   END_RUNG
   RUNG wire#powerrail
      Contact( "T-30.00_DB".ChiliAwet_3.V_CMD )
      Contact( "T-04.01_DB".Actuator.AV_Outlet )
   END_RUNG wire#w1
   RUNG wire#powerrail
      Contact( "T-04.01_DB".Cmd.Flushing )
      Contact( "T-04.01_DB".State.Flush_selected.%X2 )
   END_RUNG wire#w1
   RUNG wire#powerrail
      I_Contact( "ZSC-30.11" )
      Contact( #"AV-30.11".QCMD_OP )
   END_RUNG wire#w2
   RUNG wire#powerrail
      Contact( "ZSC-30.11" )
   END_RUNG wire#w3
   RUNG wire#powerrail
      I_Contact( #"AV-30.11".QCMD_OP )
   END_RUNG wire#w3
   // the same network as SCL:
   #"AV-30.11"(LOCK := #lock,   // "Valve"
               LIOP_SEL := #Init,
               L_AUT := #Init,
               L_REMOTE := #Init,
               L_RESET := #Reset,
               AUT_OP := ("T-30.00_DB".ChiliAwet_3.V_CMD AND "T-04.01_DB".Actuator.AV_Outlet) OR ("T-04.01_DB".Cmd.Flushing AND "T-04.01_DB".State.Flush_selected.%X2),
               FB_OPEN := NOT "ZSC-30.11" AND #"AV-30.11".QCMD_OP,
               FB_CLOSE := "ZSC-30.11" OR NOT #"AV-30.11".QCMD_OP,
               L_MON := #Init,
               INSTANCE := 'AV-30.11',
               QCMD_OP => "AV-30.11");
END_REGION

REGION Network 76: AV-30.12
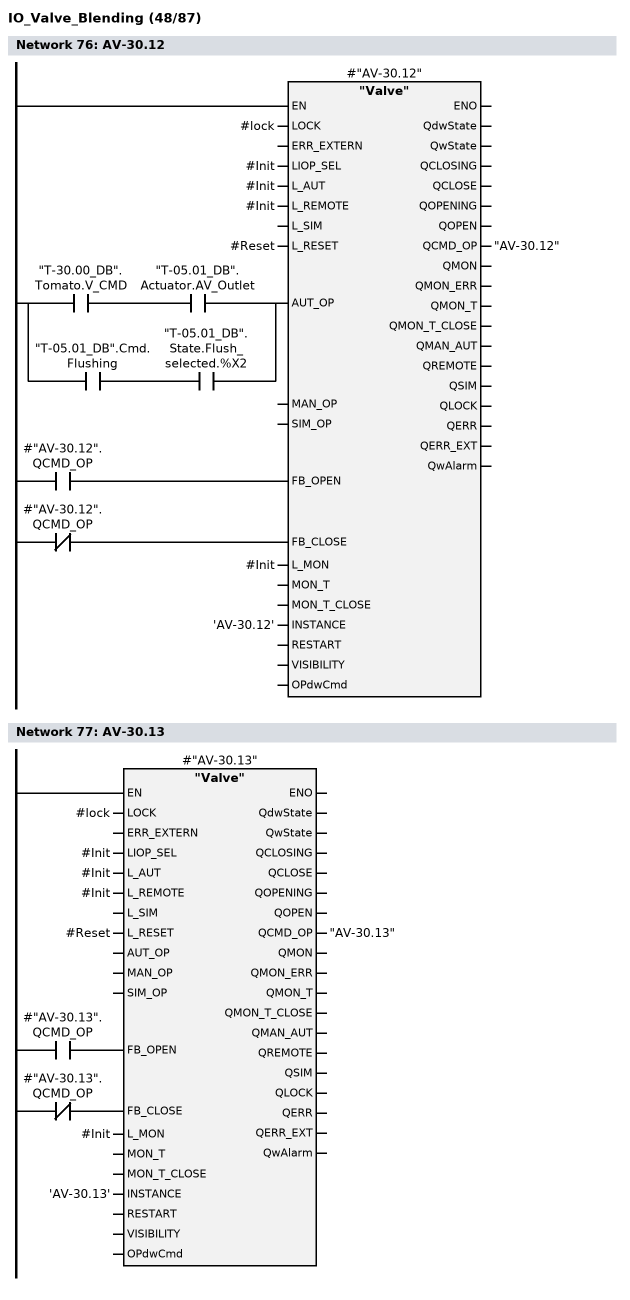
   RUNG wire#powerrail
      #"AV-30.12"(AUT_OP := wire#w1, FB_OPEN := wire#w2, FB_CLOSE := wire#w3, LOCK := #lock, ERR_EXTERN :=, LIOP_SEL := #Init, L_AUT := #Init, L_REMOTE := #Init, L_SIM :=, L_RESET := #Reset, MAN_OP :=, SIM_OP :=, L_MON := #Init, MON_T :=, MON_T_CLOSE :=, INSTANCE := 'AV-30.12', RESTART :=, VISIBILITY :=, OPdwCmd :=, QdwState =>, QwState =>, QCLOSING =>, QCLOSE =>, QOPENING =>, QOPEN =>, QCMD_OP => "AV-30.12", QMON =>, QMON_ERR =>, QMON_T =>, QMON_T_CLOSE =>, QMAN_AUT =>, QREMOTE =>, QSIM =>, QLOCK =>, QERR =>, QERR_EXT =>, QwAlarm =>)
   END_RUNG
   RUNG wire#powerrail
      Contact( "T-30.00_DB".Tomato.V_CMD )
      Contact( "T-05.01_DB".Actuator.AV_Outlet )
   END_RUNG wire#w1
   RUNG wire#powerrail
      Contact( "T-05.01_DB".Cmd.Flushing )
      Contact( "T-05.01_DB".State.Flush_selected.%X2 )
   END_RUNG wire#w1
   RUNG wire#powerrail
      Contact( #"AV-30.12".QCMD_OP )
   END_RUNG wire#w2
   RUNG wire#powerrail
      I_Contact( #"AV-30.12".QCMD_OP )
   END_RUNG wire#w3
   // the same network as SCL:
   #"AV-30.12"(LOCK := #lock,   // "Valve"
               LIOP_SEL := #Init,
               L_AUT := #Init,
               L_REMOTE := #Init,
               L_RESET := #Reset,
               AUT_OP := ("T-30.00_DB".Tomato.V_CMD AND "T-05.01_DB".Actuator.AV_Outlet) OR ("T-05.01_DB".Cmd.Flushing AND "T-05.01_DB".State.Flush_selected.%X2),
               FB_OPEN := #"AV-30.12".QCMD_OP,
               FB_CLOSE := NOT #"AV-30.12".QCMD_OP,
               L_MON := #Init,
               INSTANCE := 'AV-30.12',
               QCMD_OP => "AV-30.12");
END_REGION

REGION Network 77: AV-30.13
   RUNG wire#powerrail
      #"AV-30.13"(FB_OPEN := wire#w1, FB_CLOSE := wire#w2, LOCK := #lock, ERR_EXTERN :=, LIOP_SEL := #Init, L_AUT := #Init, L_REMOTE := #Init, L_SIM :=, L_RESET := #Reset, AUT_OP :=, MAN_OP :=, SIM_OP :=, L_MON := #Init, MON_T :=, MON_T_CLOSE :=, INSTANCE := 'AV-30.13', RESTART :=, VISIBILITY :=, OPdwCmd :=, QdwState =>, QwState =>, QCLOSING =>, QCLOSE =>, QOPENING =>, QOPEN =>, QCMD_OP => "AV-30.13", QMON =>, QMON_ERR =>, QMON_T =>, QMON_T_CLOSE =>, QMAN_AUT =>, QREMOTE =>, QSIM =>, QLOCK =>, QERR =>, QERR_EXT =>, QwAlarm =>)
   END_RUNG
   RUNG wire#powerrail
      Contact( #"AV-30.13".QCMD_OP )
   END_RUNG wire#w1
   RUNG wire#powerrail
      I_Contact( #"AV-30.13".QCMD_OP )
   END_RUNG wire#w2
   // the same network as SCL:
   #"AV-30.13"(LOCK := #lock,   // "Valve"
               LIOP_SEL := #Init,
               L_AUT := #Init,
               L_REMOTE := #Init,
               L_RESET := #Reset,
               FB_OPEN := #"AV-30.13".QCMD_OP,
               FB_CLOSE := NOT #"AV-30.13".QCMD_OP,
               L_MON := #Init,
               INSTANCE := 'AV-30.13',
               QCMD_OP => "AV-30.13");
END_REGION

REGION Network 78: AV-30.14
